(* IEC 61131-3 sources: elnaProjects/ElpcLogic/PomarKc7Changed/build_USO_ecl (part 7) *)

  fb_timer240(StrPh:=timer240);
  fb_PnmMore50(StrPh:=pmsMore50);
  fb_PnsOn(StrPh:=pnsOn, IM := Im.pns);
  fb_PmsMore300(StrPh:=pmsMore300);
  fb_Protection_Pms(StrPh:=Protection_Pms);
  fb_Error_Alg(StrPh:=Error_Alg);

  StrAlg.CanRun := StrAlg.inCanRun;
  StrAlg.OpcCommandsDisabled := StrAlg.inOpcCommandsDisabled;

  IF StrAlg.isRuning THEN

      StrAlg.hasError := pnsOn.error;

      (* не взведены защиты - запуск таймера *)
      IF NOT Protection_Pms.top THEN
  	runPhase(timer240);
      END_IF;

      (* не начался запуск пнс - запуск пнс *)
      IF NOT pnsOn.start THEN
  	runPhase(pnsOn);
      END_IF;

      (* запуск пнс завершен - запус защит *)
      IF pnsOn.top THEN
           runPhase(pmsMore50);
           runPhase(pmsMore300);
      END_IF;

      (* не завершился запуск защиты 50 - проверка давления 50 *)
      IF pmsMore50.start AND (NOT pmsMore50.top) THEN
  	IF ai.Pmaslo_sm_nizkoe.interval = _statusAi.NORMAL AND ai.Pmaslo_sm_nizkoe.value > 50.0  THEN
  	   pmsMore50.top := TRUE;
            END_IF;
      END_IF;

      (* не завершился запуск защиты 300 - проверка давления 300 *)
      IF  pmsMore300.start AND (NOT pmsMore300.top) THEN
  	IF ai.Pmaslo_sm_vysokoe.interval = _statusAi.NORMAL AND ai.Pmaslo_sm_vysokoe.value > 300.0  THEN
  	    pmsMore300.top := TRUE;
  	END_IF;
      END_IF;

      (* давление было проверено - запуск защит *)
      IF pmsMore50.top AND pmsMore300.top THEN
          runPhase(Protection_Pms);
      END_IF;

      (* запуск защит не завршен - запуск защит *)
      IF Protection_Pms.start AND (NOT Protection_Pms.top) THEN
  	runAiProtection(protections.Pmaslo_sm_nizkoe);
            runAiProtection(protections.Pmaslo_sm_vysokoe);
            Protection_Pms.top := TRUE;
      END_IF;

      (* таймер завершился до запуска защит - ошибка *)
      IF timer240.top THEN
          Error_Alg.ERROR := TRUE; (*не понятное куда его сунуть и нужен ли он*)
      ELSE
          Error_Alg.ERROR := FALSE;
      END_IF;

      (* защиты выствалены до завршения таймера - сброс таймера *)
      IF Protection_Pms.top THEN
  	resetPhase(timer240);
      END_IF;

      StrAlg.isEnded:= pnsOn.Top AND Protection_Pms.Top (*Как будто нужно таймер *);
  END_IF;

  StrAlg.CanRun := StrAlg.inCanRun;
  StrAlg.OpcCommandsDisabled := StrAlg.inOpcCommandsDisabled;

  (* ---- Если управление с ВУ заблокировано, то  передаем команду из алгоритма ---- *)
  IF StrAlg.inOpcCommandsDisabled THEN
  	StrAlg.inCommand := StrAlg.inCommand_Alg;
  ELSE (* иначе передаем команду с АРМа*)
  	StrAlg.inCommand := StrAlg.inCommand_ARM;
  END_IF;

  _sunpackerCommand(command := StrAlg.inCommand);
  	source := _sunpackerCommand.source;
  	cmd := _sunpackerCommand.cmd;

  IF cmd <> 0 AND lastCmd <> cmd AND (((NOT StrAlg.opcCommandsDisabled) AND source > 0) OR source = 0) then
  	CASE BYTE_TO_INT(cmd) OF
  		(*cmdRun*) 1: 	IF (StrAlg.CanRun) THEN
  					StrAlg.isRuning := TRUE;
  					StrAlg.isEnded := FALSE;
  					StrAlg.hasError := FALSE;
  					(*****************       OnRun       *****************)
                                                    algManager.nMode:=ModeGpa.MODE_PUSK_FIRST_FAZA1;

                                                    runPhase(pnsOn);
                                                    resetAiProtection(protections.Pmaslo_sm_nizkoe);
                                                    resetAiProtection(protections.Pmaslo_sm_vysokoe);

  					cmd_for_Status := cmd;
  					source_for_Status := source;
  					command_error_for_Status := 0;
  				ELSE
  					StrAlg.isRuning := FALSE;
  					StrAlg.isEnded := FALSE;
  					StrAlg.hasError := FALSE;

  					cmd_for_Status := 0;
  					source_for_Status := source;
  					command_error_for_Status := cmd;
  				END_IF;
  		(*cmdReset*) 2: 	StrAlg.isRuning := FALSE;
  				StrAlg.isEnded := FALSE;
  				StrAlg.hasError 	:= FALSE;

                                           (*****************       OnReset       *****************)
                                          waitReset(IN:=FALSE);
                                          StrAlg.inCanRun:=FALSE;

                                          resetPhase(timer240);
                                          resetPhase(pmsMore50);
                                          resetPhase(pnsOn);
                                          resetPhase(pmsMore300);
                                          resetPhase(Protection_Pms);
                                          resetPhase(Error_Alg);

                                          StrAlg.inOpcCommandsDisabled:=FALSE;

  				cmd_for_Status := cmd;
  				source_for_Status := source;
  				command_error_for_Status := 0;
  	END_CASE;
  	resetCmdTimer(IN := false);
  	resetCmdTimerPriznak := TRUE;
  END_IF;
  lastCmd := cmd;

  resetCmdTimer(IN := resetCmdTimerPriznak, PT := T#5S);
  IF resetCmdTimer.Q THEN
  	resetCmdTimerPriznak := FALSE;
  	source_for_Status := 0;
  	cmd_for_Status := 0;
  	command_error_for_Status := 0;
  END_IF;

  StrAlg.Start:= timer240.startStatus
              OR pmsMore50.startStatus
              OR pnsOn.startStatus
              OR Error_Alg.startStatus
              OR pmsMore300.startStatus
              OR Protection_Pms.startStatus;

  StrAlg.Error := timer240.errorStatus
              OR pmsMore50.errorStatus
              OR pnsOn.errorStatus
              OR Error_Alg.errorStatus
              OR pmsMore300.errorStatus
              OR Protection_Pms.errorStatus;

  StrAlg.Top := timer240.topStatus
              OR pmsMore50.topStatus
              OR pnsOn.topStatus
              OR Error_Alg.topStatus
              OR pmsMore300.topStatus
              OR Protection_Pms.topStatus;

  (*TODO: TYPE PROGRAM CODE HERE*)
  StrAlg.status :=  SHL(BYTE_TO_DWORD(source_for_Status), 29)
  			OR SHL(BYTE_TO_DWORD(cmd_for_Status), 26)
  			OR SHL(BYTE_TO_DWORD(command_error_for_Status), 23)
  			OR SHL(BOOL_TO_DWORD(StrAlg.OpcCommandsDisabled ), 21)
  			OR SHL(BOOL_TO_DWORD(StrAlg.hasError),4)
  			OR SHL(BOOL_TO_DWORD(StrAlg.CanRun),2)
  			OR SHL(BOOL_TO_DWORD(StrAlg.isEnded),1)
  			OR BOOL_TO_DWORD(StrAlg.isRuning);
END_FUNCTION_BLOCK

FUNCTION_BLOCK Prov_PMS
  VAR_IN_OUT
    StrAlg : struct_Alg;
  END_VAR
  VAR
    pnsOff : struct_PhaseAlgoritm;
    timer120 : struct_PhaseAlgoritm;
    Pms_less_25 : struct_PhaseAlgoritm;
    Pms_less_250 : struct_PhaseAlgoritm;
    Error_Alg : struct_PhaseAlgoritm;
    fb_Pms_less_25 : fb_ph_algoritm;
    fb_Pms_less_250 : fb_ph_algoritm;
    fb_pnsOff : fb_ph_Switch;
    fb_timer120 : fb_ph_Timer;
    fb_Error_Alg : fb_ph_algoritm;
    onInit : BOOL;
  END_VAR
  VAR_EXTERNAL
    Im : ImConfig;
    ai : AiConfig;
  END_VAR
  VAR
    _sunpackerCommand : fb_sunpackerCommand;
    source : BYTE;
    cmd : BYTE;
    _statusDualInput : TYPE_statusDualInput;
    lastCmd : BYTE;
    _Answers : TYPE_Answers;
  END_VAR
  VAR_EXTERNAL
    ModeGpa : TYPE_ModeGpa;
    algManager : struct_AlgoritmsManager;
  END_VAR
  VAR
    cmd_for_Status : BYTE;
    source_for_Status : BYTE;
    command_error_for_Status : BYTE;
    resetCmdTimer : TON;
    waitReset : TON;
    resetCmdTimerPriznak : BOOL;
    _statusAi : TYPE_StatusAi;
  END_VAR

  IF NOT onInit THEN
      fb_pnsOff(phaseNumber:=1, act:=_off);
      fb_timer120(phaseNumber:=2, delay:=T#120S);
      fb_Pms_less_25(phaseNumber:=3);
      fb_Pms_less_250(phaseNumber:=4);
      fb_Error_Alg(phaseNumber:=5);
      onInit:=TRUE;
  END_IF;

  fb_pnsOff(StrPh:=pnsOff, Im:=Im.pns);
  fb_timer120(StrPh:=timer120);
  fb_Pms_less_25(StrPh:=Pms_less_25);
  fb_Pms_less_250(StrPh:=Pms_less_250);
  fb_Error_Alg(StrPh:=Error_Alg);

  StrAlg.CanRun := StrAlg.inCanRun;
  StrAlg.OpcCommandsDisabled := StrAlg.inOpcCommandsDisabled;

  IF StrAlg.isRuning THEN
     (*IF NOT pnsOff.start THEN
  	    PNS_OFF_Ask.ask ();
      END_IF;
      IF	(PNS_OFF_Ask.answer=Answers.ANS_YES) THEN
  	    runPhase(pnsOff);
          PNS_OFF_Ask.reset ();
  	    IF NOT (Pms_less_250.top AND Pms_less_25.top) THEN
  	    	runPhase(timer120);
  	    END_IF;
      END_IF;*)

      (*запуск проверок давления*)
      IF	pnsOff.top  THEN
          runPhase(Pms_less_25);
  	    runPhase(Pms_less_250);
      END_IF;

      (*проверка давления масла низкое*)
      IF	Pms_less_25.start AND NOT Pms_less_25.top THEN
  	    IF 	ai.Pmaslo_sm_nizkoe.interval>=_statusAi.NORMAL AND ai.Pmaslo_sm_nizkoe.value < 25.0 THEN
  	  	    Pms_less_25.top:=TRUE;
  	    END_IF;
      END_IF;

      IF	Pms_less_250.start AND NOT Pms_less_250.top THEN
  	    IF	ai.Pmaslo_sm_vysokoe.interval>=_statusAi.NORMAL AND ai.Pmaslo_sm_vysokoe.value < 250.0 THEN
  	  	    Pms_less_250.top:=TRUE;
  	    END_IF;
      END_IF;

      (*ошибка заврешия алгоритма по таймеру*)
      IF	timer120.top THEN
  	    Error_Alg.ERROR := TRUE;
      ELSE
  	    Error_Alg.ERROR := FALSE;
      END_IF;

      (*если проверка прошла - сброс таймера *)
      IF	Pms_less_250.top AND Pms_less_25.top  THEN
          resetPhase(timer120);
      END_IF;
  END_IF;

  _sunpackerCommand(command := StrAlg.inCommand);
  	source := _sunpackerCommand.source;
  	cmd := _sunpackerCommand.cmd;

  IF cmd <> 0 AND lastCmd <> cmd AND (((NOT StrAlg.opcCommandsDisabled) AND source > 0) OR source = 0) then
  	CASE BYTE_TO_INT(cmd) OF
  		(*cm dRun*) 1: 	IF (StrAlg.CanRun) THEN
  					StrAlg.isRuning := TRUE;
  					StrAlg.isEnded := FALSE;
  					StrAlg.hasError := FALSE;
  					(*****************       OnRun       *****************)
                                                    algManager.nMode:=ModeGpa.MODE_PUSK_FIRST_FAZA2;

                                                    (*runPhase(timer120);
                                                    runPhase(timer5);
                                                    runPhase(Shup);
                                                    resetAiProtection(protections.dPmaslo_gaz);
                                                    resetDiProtection(protections.dPmaslo_gaz_less100);*)

  					cmd_for_Status := cmd;
  					source_for_Status := source;
  					command_error_for_Status := 0;
  				ELSE
  					StrAlg.isRuning := FALSE;
  					StrAlg.isEnded := FALSE;
  					StrAlg.hasError := FALSE;

  					cmd_for_Status := 0;
  					source_for_Status := source;
  					command_error_for_Status := cmd;
  				END_IF;
  		(*cmdReset*) 2: 	StrAlg.isRuning := FALSE;
  				StrAlg.isEnded := FALSE;
  				StrAlg.hasError 	:= FALSE;

                                           (*****************       OnReset       *****************)
                                          waitReset(IN:=FALSE);
                                          StrAlg.inCanRun:=FALSE;

                                          (*resetPhase(timer5);
                                          resetPhase(Shup);
                                          resetPhase(timer120);
                                          resetPhase(Net_Chast);
                                          resetPhase(mvOn);
                                          resetPhase(pGNSmore04);
                                          resetPhase(gotov_K_zagruzke);
                                          resetPhase(dPmg_Top);
                                          resetPhase(AutoPNS_Start);*)

                                          StrAlg.inOpcCommandsDisabled:=FALSE;

  				cmd_for_Status := cmd;
  				source_for_Status := source;
  				command_error_for_Status := 0;
  	END_CASE;
  	resetCmdTimer(IN := false);
  	resetCmdTimerPriznak := TRUE;
  END_IF;
  lastCmd := cmd;

  resetCmdTimer(IN := resetCmdTimerPriznak, PT := T#5S);
  IF resetCmdTimer.Q THEN
  	resetCmdTimerPriznak := FALSE;
  	source_for_Status := 0;
  	cmd_for_Status := 0;
  	command_error_for_Status := 0;
  END_IF;

  StrAlg.Start:= pnsOff.startStatus
              OR timer120.startStatus
              OR Pms_less_25.startStatus
              OR Pms_less_250.startStatus;

  StrAlg.Top :=  pnsOff.topStatus
              OR timer120.topStatus
              OR Pms_less_25.topStatus
              OR Pms_less_250.topStatus;

  StrAlg.Error :=  pnsOff.errorStatus
              OR timer120.errorStatus
              OR Pms_less_25.errorStatus
              OR Pms_less_250.errorStatus;

  (*TODO: TYPE PROGRAM CODE HERE*)
  StrAlg.status :=  SHL(BYTE_TO_DWORD(source_for_Status), 29)
  			OR SHL(BYTE_TO_DWORD(cmd_for_Status), 26)
  			OR SHL(BYTE_TO_DWORD(command_error_for_Status), 23)
  			OR SHL(BOOL_TO_DWORD(StrAlg.OpcCommandsDisabled ), 21)
  			OR SHL(BOOL_TO_DWORD(StrAlg.hasError),4)
  			OR SHL(BOOL_TO_DWORD(StrAlg.CanRun),2)
  			OR SHL(BOOL_TO_DWORD(StrAlg.isEnded),1)
  			OR BOOL_TO_DWORD(StrAlg.isRuning);
END_FUNCTION_BLOCK

FUNCTION_BLOCK Prov_opressovka
  VAR_IN_OUT
    StrAlg : struct_Alg;
  END_VAR
  VAR
    OPC_Control : struct_PhaseAlgoritm;
    Pms_more_50 : struct_PhaseAlgoritm;
    Pms_more_300 : struct_PhaseAlgoritm;
    dPmg_more_100 : struct_PhaseAlgoritm;
    P_zad : struct_PhaseAlgoritm;
    kran5Open : struct_PhaseAlgoritm;
    kran4Open : struct_PhaseAlgoritm;
    kran5Close : struct_PhaseAlgoritm;
    kran4Close : struct_PhaseAlgoritm;
    timer10 : struct_PhaseAlgoritm;
    P_vh_vyh_more_zad : struct_PhaseAlgoritm;
    Zapoln_Norm : struct_PhaseAlgoritm;
    First_Step : struct_PhaseAlgoritm;
    MaxZapolnenie_izm : REAL;
    Opressovka_Start : struct_Question;
    PNS_NU_ON_Ask : struct_Question;
    Zapolnit_kontur : struct_Question;
    fb_OPC_Control : fb_ph_algoritm;
    fb_Pms_more_50 : fb_ph_algoritm;
    fb_Pms_more_300 : fb_ph_algoritm;
    fb_dPmg_more_100 : fb_ph_algoritm;
    fb_P_zad : fb_ph_algoritm;
    fb_kran5Open : fb_ph_Kran;
    fb_kran4Open : fb_ph_Kran;
    fb_kran5Close : fb_ph_Kran;
    fb_kran4Close : fb_ph_Kran;
    fb_timer10 : fb_ph_Timer;
    fb_P_vh_vyh_more_zad : fb_ph_algoritm;
    fb_Zapoln_Norm : fb_ph_algoritm;
    fb_First_Step : fb_ph_algoritm;
    fb_Opressovka_Start : fb_Question;
    fb_PNS_NU_ON_Ask : fb_Question;
    fb_Zapolnit_kontur : fb_Question;
    onInit : BOOL;
  END_VAR
  VAR_EXTERNAL
    Im : ImConfig;
    ai : AiConfig;
  END_VAR
  VAR
    _sunpackerCommand : fb_sunpackerCommand;
    source : BYTE;
    cmd : BYTE;
    _statusDualInput : TYPE_statusDualInput;
    lastCmd : BYTE;
    _Answers : TYPE_Answers;
  END_VAR
  VAR_EXTERNAL
    ModeGpa : TYPE_ModeGpa;
    algManager : struct_AlgoritmsManager;
  END_VAR
  VAR
    cmd_for_Status : BYTE;
    source_for_Status : BYTE;
    command_error_for_Status : BYTE;
    resetCmdTimer : TON;
    waitReset : TON;
    resetCmdTimerPriznak : BOOL;
    _statusAi : TYPE_StatusAi;
    protections : ProtectionsConfig;
  END_VAR

  IF NOT onInit THEN
      fb_OPC_Control(phaseNumber:=1);
      fb_Pms_more_50(phaseNumber:=2);
      fb_Pms_more_300(phaseNumber:=3);
      fb_dPmg_more_100(phaseNumber:=4);
      fb_P_zad(phaseNumber:=5);
      fb_kran5Open(phaseNumber:=6, act:=_on);
      fb_kran4Open(phaseNumber:=7, act:=_on);
      fb_kran5Close(phaseNumber:=8, act:=_off);
      fb_kran4Close(phaseNumber:=9, act:=_off);
      fb_timer10(phaseNumber:=10, delay:=T#10S);
      fb_P_vh_vyh_more_zad(phaseNumber:=11);
      fb_Zapoln_Norm(phaseNumber:=12);
      fb_First_Step(phaseNumber:=13);
      Opressovka_Start.AnswerVariants:=_Answers.ANS_YES + _Answers.ANS_NO;
      PNS_NU_ON_Ask.AnswerVariants:=_Answers.ANS_YES;
      Zapolnit_kontur.AnswerVariants:=_Answers.ANS_YES;
      onInit:=TRUE;
  END_IF;

  fb_OPC_Control(StrPh:=OPC_Control);
  fb_Pms_more_50(StrPh:=Pms_more_50);
  fb_Pms_more_300(StrPh:=Pms_more_300);
  fb_dPmg_more_100(StrPh:=dPmg_more_100);
  fb_P_zad(StrPh:=P_zad);
  fb_kran5Open(StrPh:=kran5Open, Im:=Im.Kran5);
  fb_kran4Open(StrPh:=kran4Open, Im:=Im.Kran4);
  fb_kran5Close(StrPh:=kran5Close, Im:=Im.Kran5);
  fb_kran4Close(StrPh:=kran4Close, Im:=Im.Kran4);
  fb_timer10(StrPh:=timer10);
  fb_P_vh_vyh_more_zad(StrPh:=P_vh_vyh_more_zad);
  fb_Zapoln_Norm(StrPh:=Zapoln_Norm);
  fb_First_Step(StrPh:=First_Step);
  fb_Opressovka_Start(StrQ:=Opressovka_Start);
  fb_PNS_NU_ON_Ask(StrQ:=PNS_NU_ON_Ask);
  fb_Zapolnit_kontur(StrQ:=Zapolnit_kontur);

  StrAlg.CanRun := StrAlg.inCanRun;
  StrAlg.OpcCommandsDisabled := StrAlg.inOpcCommandsDisabled;

  IF StrAlg.isRuning THEN
     (*IF	algManager.mode <> ModeGpa.MODE_O THEN
  	    askQuestion(Opressovka_Start);
      END_IF;*)

      IF	Opressovka_Start.answer=_Answers.ANS_YES THEN
  	    askQuestion(Opressovka_Start);
  	    Im.kran6.inOpcCommandsDisabled := FALSE;
  	    (*algManager.setMode(nMode:=ModeGpa.MODE_O);*)
  	    runPhase(OPC_Control);
  	    resetAiProtection(protections.Pgaza_na_vyhode_nagnetatelia_GPA_STOP);
  	    resetAiProtection(protections.Pgaza_na_vhode_nagnetatelia_GPA_STOP);
          ELSIF Opressovka_Start.answer=_Answers.ANS_no THEN
                resetQuestion(Opressovka_Start);
      END_IF;

      IF	OPC_Control.start AND NOT OPC_Control.top THEN
  	    askQuestion(PNS_NU_ON_Ask);
      END_IF;
      IF	(PNS_NU_ON_Ask.answer=_Answers.ANS_YES) AND NOT OPC_Control.top THEN
  	    OPC_Control.top:=TRUE;
  	    resetQuestion(PNS_NU_ON_Ask);
      END_IF;

      IF	OPC_Control.top AND NOT Pms_more_50.start  THEN
  	    Im.pns.inOpcCommandsDisabled := FALSE;
  	    Im.kran6.inOpcCommandsDisabled := FALSE;
  	    runPhase(Pms_more_50);
  	    runPhase(Pms_more_300);
      END_IF;
      IF	OPC_Control.top AND Im.pns.onStatus = _statusDualInput.STATUS_On AND NOT dPmg_more_100.start THEN
  	    Im.nu1.inOpcCommandsDisabled := FALSE;
  	    Im.nu2.inOpcCommandsDisabled := FALSE;
  	    runPhase(dPmg_more_100);
      END_IF;

      IF	Im.nu1.onStatus = _statusDualInput.STATUS_On OR Im.nu2.onStatus = _statusDualInput.STATUS_On AND dPmg_more_100.start AND NOT dPmg_more_100.top THEN
  	    IF ai.dPmaslo_gaz.interval	>=	_statusAi.NORMAL AND
  		    ai.dPmaslo_gaz.value > 150.0 AND Im.SingleSignals.dP_maslo_gaz_Less100.reliability = TRUE AND NOT Im.SingleSignals.dP_maslo_gaz_Less100.Q THEN
  		    dPmg_more_100.top:=TRUE;
  		    runAiProtection(protections.dPmaslo_gaz);
  		    runDiProtection(protections.dPmaslo_gaz_less100);
  	    END_IF;
      END_IF;

      IF	Im.pns.onStatus = _statusDualInput.STATUS_On AND Pms_more_50.start AND NOT Pms_more_50.top THEN
  	        IF	ai.Pmaslo_sm_nizkoe.interval	>=	_statusAi.NORMAL AND
  		        ai.Pmaslo_sm_nizkoe.value > 50.0 THEN
  		        Pms_more_50.top:=TRUE;
                  runAiProtection(protections.Pmaslo_sm_nizkoe);
  	    END_IF;
      END_IF;

      IF	Im.pns.onStatus = _statusDualInput.STATUS_On AND Pms_more_300.start AND NOT Pms_more_300.top THEN
  	    IF	ai.Pmaslo_sm_vysokoe.interval	>=	_statusAi.NORMAL AND
  		    ai.Pmaslo_sm_vysokoe.value > 300.0 THEN
  		    Pms_more_300.top:=TRUE;
  		    runAiProtection(protections.Pmaslo_sm_vysokoe);
  	    END_IF;
      END_IF;

      (*IF	dPmg_more_100.top AND Pms_more_50.top AND Pms_more_300.top THEN
  	    CASE	Auto.value OF
  	    0:	Im.kran3.inOpcCommandsDisabled := FALSE;
  		Im.kran4.inOpcCommandsDisabled := FALSE;
  		Im.kran5.inOpcCommandsDisabled := FALSE;
  		Im.kran3b.inOpcCommandsDisabled := FALSE;
  		resetPhase(Zapolnit_kontur);
  		IF	Im.PerepadDavlenieKran1_Less100.Q THEN
  			Im.kran1.inOpcCommandsDisabled := FALSE;
  			Im.kran2.inOpcCommandsDisabled := FALSE;
  		ELSE
  			Im.kran1.inOpcCommandsDisabled := TRUE;
  			Im.kran2.inOpcCommandsDisabled := TRUE;
  		END_IF
  		resetPhase(P_vh_vyh_more_zad);
  		resetPhase(kran5Open);
  		resetPhase(kran4Open);
  		resetPhase(timer10);
  		resetPhase(kran5Close);
  		resetPhase(P_zad);
  		resetPhase(First_Step);
  		resetPhase(kran4Close);
  		(*MaxZapolnenie_izm:=0;
  		MaxZapolnenie.setValue (0);
  	1:
  		Zapoln_Norm.top:= MaxZapolnenie.value - MaxZapolnenie_izm > 0.4 AND MaxZapolnenie.value >= 0.4 AND MaxZapolnenie.value <= 10 AND
  			ai.DGazaNaVhodeNagnetatelja.interval >= _statusAi.NORMAL AND MaxZapolnenie.value - ai.DGazaNaVhodeNagnetatelja.value > 0.4 AND
  			ai.DGazaNaVyhodeNagnetatelja.interval >= _statusAi.NORMAL AND MaxZapolnenie.value - ai.DGazaNaVyhodeNagnetatelja.value > 0.4 *)
  		IF	kran4Close.top AND Zapoln_Norm.top AND NOT P_zad.start THEN
  			resetPhase(P_vh_vyh_more_zad);
  			resetPhase(kran5Open);
  			resetPhase(kran4Open);
  			resetPhase(timer10);
  			resetPhase(kran5Close);
  			resetPhase(kran4Close);
  		END_IF;
  		IF	NOT kran4Close.top OR kran4Close.top AND Zapoln_Norm.top AND NOT P_zad.start THEN
  		 	runPhase(P_zad);
  		END_IF;
  		IF NOT P_zad.top AND P_zad.start AND Zapoln_Norm.top THEN
  			askQuestion(Zapolnit_kontur);
  			Im.kran3.inOpcCommandsDisabled := TRUE;
  			Im.kran4.inOpcCommandsDisabled := TRUE;
  			Im.kran5.inOpcCommandsDisabled := TRUE;
  			Im.kran3b.inOpcCommandsDisabled := TRUE;
  			Im.kran1.inOpcCommandsDisabled := TRUE;
  			Im.kran2.inOpcCommandsDisabled := TRUE;

  		ELSIF NOT Zapoln_Norm.top AND NOT P_zad.top THEN
  				resetQuestion(Zapolnit_kontur);
  		END_IF;

          IF	(Zapolnit_kontur.answer=_Answers.ANS_YES) AND P_zad.start THEN
  			(*MaxZapolnenie_izm:= MaxZapolnenie.value;*)
  			IF 	NOT First_Step.top THEN
  				runPhase(kran5Open);
  			ELSE
  				runPhase(kran4Open);
  			END_IF;
  			resetQuestion(Zapolnit_kontur);
  			P_zad.top:=TRUE;
  		END_IF;
                      (*

  		IF	P_zad.top AND NOT kran4Close.top THEN
  			MaxZapolnenie.newvalue:=MaxZapolnenie_izm;
  		ELSE
  			MaxZapolnenie.newvalue:= MaxZapolnenie.newvalue;
  		END_IF;*)

  		IF	kran5Open.top AND NOT First_Step.top THEN
  			runPhase(kran4Open);
  		END_IF;

          IF 	kran4Open.top AND NOT timer10.top AND NOT First_Step.top THEN
  			runPhase(timer10);
  		END_IF;

  		IF	timer10.top AND NOT First_Step.top THEN
  			runPhase(kran5Close);
  		END_IF;

  		IF	kran5Close.top OR First_Step.top AND kran4Open.top THEN
  			runPhase(P_vh_vyh_more_zad);
          END_IF;

  		IF	ai.Pgaza_na_vhode_nagnetatelia.interval >= _statusAi.NORMAL (*AND ai.Pgaza_na_vhode_nagnetatelia.value >= MaxZapolnenie.value*) AND
  			ai.Pgaza_na_vyhode_nagnetatelia.interval >= _statusAi.NORMAL (*AND ai.Pgaza_na_vyhode_nagnetatelia.value >= MaxZapolnenie.value*) AND  P_vh_vyh_more_zad.start AND NOT P_vh_vyh_more_zad.top THEN
  			runPhase(kran4Close);
  			P_vh_vyh_more_zad.top:=TRUE;
  		END_IF;

  		IF	kran4Close.top THEN
  			First_Step.top:=TRUE;
  			Im.kran3.inOpcCommandsDisabled := FALSE;
  			Im.kran4.inOpcCommandsDisabled := FALSE;
  			Im.kran5.inOpcCommandsDisabled := FALSE;
  			Im.kran3b.inOpcCommandsDisabled := FALSE;

              IF	Zapoln_Norm.top THEN
  				resetPhase(P_zad);
  			END_IF;

              IF	Im.SingleSignals.dp_kran1_Less100.Q THEN
  				Im.kran1.inOpcCommandsDisabled := FALSE;
  				Im.kran2.inOpcCommandsDisabled := FALSE;
  			ELSE
  				Im.kran1.inOpcCommandsDisabled := TRUE;
  				Im.kran2.inOpcCommandsDisabled := TRUE;
  			END_IF;
  		ELSE
  			Im.kran1.inOpcCommandsDisabled := TRUE;
  			Im.kran2.inOpcCommandsDisabled := TRUE;
  	    END_IF;
          END_IF;
          (*END_CASE;
  END_IF;*)

  _sunpackerCommand(command := StrAlg.inCommand);
  	source := _sunpackerCommand.source;
  	cmd := _sunpackerCommand.cmd;

  IF cmd <> 0 AND lastCmd <> cmd AND (((NOT StrAlg.opcCommandsDisabled) AND source > 0) OR source = 0) then
  	CASE BYTE_TO_INT(cmd) OF
  		(*cm dRun*) 1: 	IF (StrAlg.CanRun) THEN
  					StrAlg.isRuning := TRUE;
  					StrAlg.isEnded := FALSE;
  					StrAlg.hasError := FALSE;
  					(*****************       OnRun       *****************)
                                                    algManager.nMode:=ModeGpa.MODE_PUSK_FIRST_FAZA2;

                                                    (*runPhase(timer120);
                                                    runPhase(timer5);
                                                    runPhase(Shup);
                                                    resetAiProtection(protections.dPmaslo_gaz);
                                                    resetDiProtection(protections.dPmaslo_gaz_less100);*)

  					cmd_for_Status := cmd;
  					source_for_Status := source;
  					command_error_for_Status := 0;
  				ELSE
  					StrAlg.isRuning := FALSE;
  					StrAlg.isEnded := FALSE;
  					StrAlg.hasError := FALSE;

  					cmd_for_Status := 0;
  					source_for_Status := source;
  					command_error_for_Status := cmd;
  				END_IF;
  		(*cmdReset*) 2: 	StrAlg.isRuning := FALSE;
  				StrAlg.isEnded := FALSE;
  				StrAlg.hasError 	:= FALSE;

                                           (*****************       OnReset       *****************)
                                          waitReset(IN:=FALSE);
                                          StrAlg.inCanRun:=FALSE;

                                          (*resetPhase(timer5);
                                          resetPhase(Shup);
                                          resetPhase(timer120);
                                          resetPhase(Net_Chast);
                                          resetPhase(mvOn);
                                          resetPhase(pGNSmore04);
                                          resetPhase(gotov_K_zagruzke);
                                          resetPhase(dPmg_Top);
                                          resetPhase(AutoPNS_Start);*)

                                          StrAlg.inOpcCommandsDisabled:=FALSE;

  				cmd_for_Status := cmd;
  				source_for_Status := source;
  				command_error_for_Status := 0;
  	END_CASE;
  	resetCmdTimer(IN := false);
  	resetCmdTimerPriznak := TRUE;
  END_IF;
  lastCmd := cmd;

  resetCmdTimer(IN := resetCmdTimerPriznak, PT := T#5S);
  IF resetCmdTimer.Q THEN
  	resetCmdTimerPriznak := FALSE;
  	source_for_Status := 0;
  	cmd_for_Status := 0;
  	command_error_for_Status := 0;
  END_IF;

  StrAlg.Start:= OPC_Control.startStatus
              OR Pms_more_50.startStatus
              OR Pms_more_300.startStatus
              OR dPmg_more_100.startStatus
              OR P_zad.startStatus
              OR kran5Open.startStatus
              OR kran4Open.startStatus
              OR kran5Close.startStatus
              OR kran4Close.startStatus
              OR timer10.startStatus
              OR P_vh_vyh_more_zad.startStatus
              OR Zapoln_Norm.startStatus
              OR First_Step.startStatus;

  StrAlg.Top :=  OPC_Control.topStatus
              OR Pms_more_50.topStatus
              OR Pms_more_300.topStatus
              OR dPmg_more_100.topStatus
              OR P_zad.topStatus
              OR kran5Open.topStatus
              OR kran4Open.topStatus
              OR kran5Close.topStatus
              OR kran4Close.topStatus
              OR timer10.topStatus
              OR P_vh_vyh_more_zad.topStatus
              OR Zapoln_Norm.topStatus
              OR First_Step.topStatus;

  StrAlg.Error :=  OPC_Control.errorStatus
              OR Pms_more_50.errorStatus
              OR Pms_more_300.errorStatus
              OR dPmg_more_100.errorStatus
              OR P_zad.errorStatus
              OR kran5Open.errorStatus
              OR kran4Open.errorStatus
              OR kran5Close.errorStatus
              OR kran4Close.errorStatus
              OR timer10.errorStatus
              OR P_vh_vyh_more_zad.errorStatus
              OR Zapoln_Norm.errorStatus
              OR First_Step.errorStatus;

  (*TODO: TYPE PROGRAM CODE HERE*)
  StrAlg.status :=  SHL(BYTE_TO_DWORD(source_for_Status), 29)
  			OR SHL(BYTE_TO_DWORD(cmd_for_Status), 26)
  			OR SHL(BYTE_TO_DWORD(command_error_for_Status), 23)
  			OR SHL(BOOL_TO_DWORD(StrAlg.OpcCommandsDisabled ), 21)
  			OR SHL(BOOL_TO_DWORD(StrAlg.hasError),4)
  			OR SHL(BOOL_TO_DWORD(StrAlg.CanRun),2)
  			OR SHL(BOOL_TO_DWORD(StrAlg.isEnded),1)
  			OR BOOL_TO_DWORD(StrAlg.isRuning);
END_FUNCTION_BLOCK

FUNCTION_BLOCK Pusk_second_faza_chastotny
  VAR_IN_OUT
    StrAlg : struct_Alg;
  END_VAR
  VAR
    timer120 : struct_PhaseAlgoritm;
    timer5 : struct_PhaseAlgoritm;
    Shup : struct_PhaseAlgoritm;
    Net_Chast : struct_PhaseAlgoritm;
    mvOn : struct_PhaseAlgoritm;
    pGNSmore04 : struct_PhaseAlgoritm;
    gotov_K_zagruzke : struct_PhaseAlgoritm;
    dPmg_Top : struct_PhaseAlgoritm;
    AutoPNS_Start : struct_PhaseAlgoritm;
    fb_timer120 : fb_ph_Timer;
    fb_timer5 : fb_ph_Timer;
    fb_Shup : fb_ph_OilPump;
    fb_Net_Chast : fb_ph_algoritm;
    fb_mvOn : fb_ph_SectionSwitch;
    fb_pGNSmore04 : fb_ph_algoritm;
    fb_gotov_K_zagruzke : fb_ph_algoritm;
    fb_dPmg_Top : fb_ph_algoritm;
    fb_AutoPNS_Start : fb_ph_algoritm;
    _sunpackerCommand : fb_sunpackerCommand;
    _statusDualInput : TYPE_statusDualInput;
    _Answers : TYPE_Answers;
    source : BYTE;
    cmd : BYTE;
    lastCmd : BYTE;
    source_for_Status : BYTE;
    cmd_for_Status : BYTE;
    command_error_for_Status : BYTE;
    resetCmdTimer : TON;
    resetCmdTimerPriznak : BOOL;
    onInit : BOOL;
    waitReset : TON;
  END_VAR
  VAR_EXTERNAL
    ModeGpa : TYPE_ModeGpa;
    algManager : struct_AlgoritmsManager;
    IM : ImConfig;
    protections : ProtectionsConfig;
    algoritms : AlgoritmsConfig;
    ai : AiConfig;
  END_VAR
  VAR
    statusAi : TYPE_StatusAi;
  END_VAR

  IF NOT onInit THEN
           fb_timer120(phaseNumber:=1, delay:=T#120S);
           fb_timer5(phaseNumber:=2, delay:=T#5S);
           fb_Shup(phaseNumber:=3);
           fb_Net_Chast(phaseNumber:=4);
           fb_mvOn(phaseNumber:=5,  act:=_on);
           fb_pGNSmore04(phaseNumber:=6);
           fb_gotov_K_zagruzke(phaseNumber:=7);
           fb_dPmg_Top(phaseNumber:=8);
           fb_AutoPNS_Start(phaseNumber:=9, act:=_run, waitCompletion:=FALSE);
  onInit:=TRUE;
  END_IF;

  fb_timer120(StrPh:=timer120);
  fb_timer5(StrPh:= timer5);
  fb_Shup(StrPh:= Shup);
  fb_Net_Chast(StrPh:=Net_Chast);
  fb_mvOn(StrPh:=mvOn, Im:=IM.mv);
  fb_pGNSmore04(StrPh:=pGNSmore04);
  fb_gotov_K_zagruzke(StrPh:=gotov_K_zagruzke);
  fb_dPmg_Top(StrPh:=dPmg_Top);
  fb_AutoPNS_Start(StrPh:=AutoPNS_Start, alg:=algoritms.autoPns);

  StrAlg.CanRun := StrAlg.inCanRun;
  StrAlg.OpcCommandsDisabled := StrAlg.inOpcCommandsDisabled;

  IF StrAlg.isRuning THEN
      (* мв не включен - запуск таймера *)
      IF NOT mvOn.top THEN
  	runphase(timer120);
      END_IF;
      (* частотный пуск не совершен - запуск таймера *)
      IF NOT Net_Chast.top THEN
  	runphase(timer5);
      END_IF;

      (* ШУП не запущен - запуск *)
      IF NOT Shup.start THEN
  	runphase(Shup);
      END_IF;

      (* ШУП не завершился - запуск ШУПб МВ *)
      IF NOT Shup.top AND Shup.start THEN
  	runIfNotRunningSO(IM.SingleOutputs.Pusk_SHUP);
  	Shup.top:=TRUE;
  	runphase(mvOn);
      END_IF;

      (* частотный пуск не запущен - запуск *)
      IF NOT Net_Chast.start THEN
  	runphase(Net_Chast);
      END_IF;

      (* частотный пуск не завершился - запуск *)
      IF Net_Chast.start AND (NOT Net_Chast.top) THEN
  	IF (NOT IM.SingleSignals.Chastotny_pusk.Q) AND (IM.SingleSignals.Chastotny_pusk.status = 1) THEN
  		Net_Chast.top:=TRUE;
  		resetPhase(timer5);
  	END_IF;
      END_IF;

      (* таймер не истек и мв не включен - вовзедение защиты *)
      IF (NOT timer120.top) AND (NOT mvOn.top) THEN
  	runDiProtection(protections.Fail_chastotnii_pusk);
      ELSE
  	resetDiProtection(protections.Fail_chastotnii_pusk);
      END_IF;

      (* мв не завершился - включение мв *)
      IF mvOn.start AND NOT mvOn.top THEN
  	IF IM.mv.onStatus = _statusDualInput.STATUS_ON THEN
                mvOn.top:=TRUE;
  	END_IF;
      END_IF;

      (* мв завершился - что-то делаем *)
      IF mvOn.top THEN
  	IF NOT pGNSmore04.start (*AND (algManager.mode = ModeGpa.MODE_PUSKPP_Ch OR algManager.mode = ModeGpa.MODE_PUSKAP_Ch)какой режим *) THEN
  		runphase(pGNSmore04);
  	END_IF;
           (* IF NOT autoAVOM_canrun_flag THEN
                algoritms.AutoAvom.CanRun:=TRUE;
  	    autoAVOM_canrun_flag:=TRUE; kto ti
  	END_IF;*)
  	resetPhase(timer120);
  	runphase(gotov_K_zagruzke);

            IF NOT dPmg_Top.start (* AND ((algManager.mode = modegpa.MODE_PUSKAP_Ch) OR (algManager.mode = modegpa.MODE_PUSKPP_Ch))*) THEN
                runphase(dPmg_Top);
  	END_IF;

            runAiProtection(protections.Pgaza_na_vyhode_nagnetatelia_GPA_STOP);
  	runDiProtection(protections.Off_avar_vikluchatel);
  	runDiProtection(protections.Reg_vozb_off);
      END_IF;

      IF dPmg_Top.start AND NOT dPmg_Top.top THEN
  	IF NOT IM.SingleSignals.dP_maslo_gaz_Less100.Q AND IM.SingleSignals.dP_maslo_gaz_Less100.status = 1 AND ai.dPmaslo_gaz.value > 150.0 THEN
  		dPmg_Top.top:=TRUE;
  		runAiProtection(protections.dPmaslo_gaz);
  		runDiProtection(protections.dPmaslo_gaz_less100);
  		resetAiProtection(protections.Pgaza_na_vhode_nagnetatelia_GPA_STOP);
  		resetAiProtection(protections.Pgaza_na_vyhode_nagnetatelia_GPA_STOP);
  		algoritms.autoNu.CanRun:=TRUE;
  		(*algoritms.autoNu.run(); кого чего, ничего не понимаю *)
  	END_IF;
      END_IF;

      IF pGNSmore04.start AND NOT pGNSmore04.top THEN
  	IF ai.Pmasla_posle_GNS.interval (*почему интервал, если есть статус *) >= statusAi.NORMAL AND ai.Pmasla_posle_GNS.value > 400.0 THEN
  	  	pGNSmore04.top:=TRUE;
  	END_IF;
      END_IF;

      IF (pGNSmore04.top AND gotov_K_zagruzke.top AND dPmg_Top.top )(*AND (algManager.mode = modegpa.MODE_PUSKAP_Ch OR (algManager.mode = modegpa.MODE_PUSKPP_Ch) *)OR
  	(gotov_K_zagruzke.top) (*AND (algManager.mode = modegpa.MODE_PUSKV_Ch OR algManager.mode = modegpa.MODE_I))*) AND NOT AutoPNS_Start.top  THEN
  	algoritms.AutoPns.CanRun :=TRUE;
  	(*algoritms.AutoPns;*)
  	AutoPNS_Start.top:=TRUE;
      END_IF;

      IF (NOT Net_Chast.top AND timer5.top) OR (timer120.top AND NOT mvOn.top) THEN
  	algoritms.ao.CanRun:=TRUE;
  	(*algoritms.ao.run ();*)
      END_IF;
  END_IF;

  StrAlg.CanRun := StrAlg.inCanRun;
  StrAlg.OpcCommandsDisabled := StrAlg.inOpcCommandsDisabled;

  (* ---- Если управление с ВУ заблокировано, то  передаем команду из алгоритма ---- *)
  IF StrAlg.inOpcCommandsDisabled THEN
  	StrAlg.inCommand := StrAlg.inCommand_Alg;
  ELSE (* иначе передаем команду с АРМа*)
  	StrAlg.inCommand := StrAlg.inCommand_ARM;
  END_IF;

  _sunpackerCommand(command := StrAlg.inCommand);
  	source := _sunpackerCommand.source;
  	cmd := _sunpackerCommand.cmd;

  IF cmd <> 0 AND lastCmd <> cmd AND (((NOT StrAlg.opcCommandsDisabled) AND source > 0) OR source = 0) then
  	CASE BYTE_TO_INT(cmd) OF
  		(*cmdRun*) 1: 	IF (StrAlg.CanRun) THEN
  					StrAlg.isRuning := TRUE;
  					StrAlg.isEnded := FALSE;
  					StrAlg.hasError := FALSE;
  					(*****************       OnRun       *****************)
                                                    algManager.nMode:=ModeGpa.MODE_PUSK_FIRST_FAZA2;

                                                    runPhase(timer120);
                                                    runPhase(timer5);
                                                    runPhase(Shup);
                                                    resetAiProtection(protections.dPmaslo_gaz);
                                                    resetDiProtection(protections.dPmaslo_gaz_less100);

  					cmd_for_Status := cmd;
  					source_for_Status := source;
  					command_error_for_Status := 0;
  				ELSE
  					StrAlg.isRuning := FALSE;
  					StrAlg.isEnded := FALSE;
  					StrAlg.hasError := FALSE;

  					cmd_for_Status := 0;
  					source_for_Status := source;
  					command_error_for_Status := cmd;
  				END_IF;
  		(*cmdReset*) 2: 	StrAlg.isRuning := FALSE;
  				StrAlg.isEnded := FALSE;
  				StrAlg.hasError 	:= FALSE;

                                           (*****************       OnReset       *****************)
                                          waitReset(IN:=FALSE);
                                          StrAlg.inCanRun:=FALSE;

                                          resetPhase(timer5);
                                          resetPhase(Shup);
                                          resetPhase(timer120);
                                          resetPhase(Net_Chast);
                                          resetPhase(mvOn);
                                          resetPhase(pGNSmore04);
                                          resetPhase(gotov_K_zagruzke);
                                          resetPhase(dPmg_Top);
                                          resetPhase(AutoPNS_Start);

                                          StrAlg.inOpcCommandsDisabled:=FALSE;

  				cmd_for_Status := cmd;
  				source_for_Status := source;
  				command_error_for_Status := 0;
  	END_CASE;
  	resetCmdTimer(IN := false);
  	resetCmdTimerPriznak := TRUE;
  END_IF;
  lastCmd := cmd;

  resetCmdTimer(IN := resetCmdTimerPriznak, PT := T#5S);
  IF resetCmdTimer.Q THEN
  	resetCmdTimerPriznak := FALSE;
  	source_for_Status := 0;
  	cmd_for_Status := 0;
  	command_error_for_Status := 0;
  END_IF;

  StrAlg.Start:= timer120.startStatus
              OR timer5.startStatus
              OR Shup.startStatus
              OR Net_Chast.startStatus
              OR mvOn.startStatus
              OR pGNSmore04.startStatus
              OR gotov_K_zagruzke.startStatus
              OR dPmg_Top.startStatus
              OR AutoPNS_Start.startStatus;

  StrAlg.Error := timer120.errorStatus
              OR timer5.errorStatus
              OR Shup.errorStatus
              OR Net_Chast.errorStatus
              OR mvOn.errorStatus
              OR pGNSmore04.errorStatus
              OR gotov_K_zagruzke.errorStatus
              OR dPmg_Top.errorStatus
              OR AutoPNS_Start.errorStatus;

  StrAlg.Top := timer120.topStatus
              OR timer5.topStatus
              OR Shup.topStatus
              OR Net_Chast.topStatus
              OR mvOn.topStatus
              OR gotov_K_zagruzke.topStatus
              OR dPmg_Top.topStatus
              OR AutoPNS_Start.topStatus
              OR pGNSmore04.topStatus;

  (*TODO: TYPE PROGRAM CODE HERE*)
  StrAlg.status :=  SHL(BYTE_TO_DWORD(source_for_Status), 29)
  			OR SHL(BYTE_TO_DWORD(cmd_for_Status), 26)
  			OR SHL(BYTE_TO_DWORD(command_error_for_Status), 23)
  			OR SHL(BOOL_TO_DWORD(StrAlg.OpcCommandsDisabled ), 21)
  			OR SHL(BOOL_TO_DWORD(StrAlg.hasError),4)
  			OR SHL(BOOL_TO_DWORD(StrAlg.CanRun),2)
  			OR SHL(BOOL_TO_DWORD(StrAlg.isEnded),1)
  			OR BOOL_TO_DWORD(StrAlg.isRuning);
END_FUNCTION_BLOCK

FUNCTION_BLOCK proc_algoritms
  VAR
    fb_RemontAlg : RemontAlg;
    fb_TestProtectionAlg : TestProtectionAlg;
    fb_TestImAlg : TestImAlg;
    fb_AutoTen : fb_AutoTenAlg;
    fb_AutoPns : fb_AutoPnsAlg;
    fb_AutoAvom : fb_AutoAvomAlg;
    fb_vibegPNS : fb_vibegPNSAlg;
    fb_AutoNU : fb_AutoNUAlg;
    fb_puskOilSystem : fb_puskOilSystemAlg;
    fb_AntiPompag : fb_AntiPompagAlg;
    fb_NOAlg : NOAlg;
    fb_AOAlg : AOAlg;
    fb_ppuALG : ppuAlg;
    fb_fillingAlg : fillingAlg;
    fb_engineRunAlg : engineRunAlg;
    fb_puskKalg : puskKalg;
    fb_puskValg : puskValg;
    fb_testdPmgAlg : testdPmgAlg;
    fb_testPmsAlg : testPmsAlg;
    fb_ApuskAlg : ApuskAlg;
    fb_SemiAutoPuskAlg : SemiAutoPuskAlg;
    fb_Pusk_first_faza1 : Pusk_first_faza1;
    fb_Pusk_first_faza2 : Pusk_first_faza2;
    fb_Pusk_third_faza : Pusk_third_faza;
    fb_Pusk_Prov_PMS : Prov_PMS;
    fb_Prov_opressovka : Prov_opressovka;
    fb_Pusk_second_faza_chastotny : Pusk_second_faza_chastotny;
    fb_Pusk_second_faza_reactor : Pusk_second_faza_reactor;
  END_VAR
  VAR_EXTERNAL
    algoritms : AlgoritmsConfig;
    AlgQuestions : AlgoritmsQuestions;
    ai : AiConfig;
    IM : ImConfig;
    AlgTimers : struct_AlgTimers;
  END_VAR

  fb_RemontAlg(StrAlg:=algoritms.Remont);

  fb_TestProtectionAlg(StrAlg:=algoritms.TestProtection);

  fb_TestImAlg(StrAlg:=algoritms.testIm);

  (*fb_AutoTen(StrAlg:= algoritms.AutoTen,
  T_masla:= ai.Toporno_podshipnika_EDT_1,
  Uroven_masla:= ai.Yroven_masla_MB,
  offTemperature:= Im.AutoTen_offTemperature,
  TEN:= Im.Ten,
  PNS:= Im.pns);*)

  (*fb_AutoPns(StrAlg:= algoritms.AutoPns,
  Poil:= ai.Pmasla_posle_GNS,
  Ust_Run:= Im.AutoPns_UstRun,
  Ust_Stop:= Im.AutoPns_UstStop,
  Nasos:= Im.pns,
  diPlow:= Im.SingleSignals.P_oil_low);*)

  (*fb_AutoAvom(StrAlg:= algoritms.AutoAvom,
  im1:= Im.v1_Avom,
  im2:= Im.v2_Avom,
  on1Temperature:= Im.AutoAvom_onTemp1,
  on2Temperature:= Im.AutoAvom_onTemp2,
  hystereses:= Im.AutoAvom_hysteresis,
  ai:= ai.Tnarujnogo_vozduha);*)

  fb_vibegPNS(StrAlg:=algoritms.vibegPNS,
  algContinue:=AlgQuestions.vibegPNS_algContinue
  );

  (*fb_AutoNU(StrAlg:=algoritms.autoNu,
  nu1:=Im.nu1,
  nu2:=Im.nu2,
  Ust_Swap:= Im.AutoNU_Ust_Swap,
  mainNU:= Im.AutoNU_mainNU,
  dPoil:=ai.Tmasla_MB,
  Lowdp_di:=Im.SingleSignals.dP_oilgaz_low
  );*)

  fb_puskOilSystem(StrAlg:=algoritms.puskOilSystem);

  (*fb_AntiPompag(StrAlg:=algoritms.AntiPompag,
  Rashod:= ai.Vibro_skorost_OP_shesterni_RED_T6,
  Zapas:= ai.Vibro_skorost_OP_shesterni_RED_T5,
  P_gasIn:=ai.dPgaza_na_maslo_filtre,
  T_gasIn:=ai.Tgaza_na_vhode_H,
  dP_konf:=ai.dPgaza_na_konfuzore,
  Kran6:= im.Kran6,
  UgolVNA:= im.AntiPompag_UgolVNA,
  K:=im.AntiPompag_K,
  A:=im.AntiPompag_A,
  y0:=im.AntiPompag_y0);*)

  fb_NOAlg(StrAlg:=algoritms.no);

  fb_AOAlg(StrAlg:=algoritms.ao);

  fb_ppuAlg(StrAlg:=algoritms.ppu);

  fb_fillingAlg(StrAlg:=algoritms.filling);

  fb_engineRunAlg(StrAlg:=algoritms.engineRun);

  fb_puskKalg(StrAlg:=algoritms.puskK,
  questionFilling:=AlgQuestions.puskK_questionFilling,
   questionUnload:=AlgQuestions.puskK_questionUnload
  );

  fb_puskValg(StrAlg:=algoritms.puskV,
   questionEngine:=AlgQuestions.puskV_questionEngine,
    questionMVoff:=AlgQuestions.puskV_questionMVoff
  );

  fb_testdPmgAlg(StrAlg:=algoritms.testdPmg,
   algContinue:=AlgQuestions.testdPmg_algContinue
  );

  fb_testPmsAlg(StrAlg:=algoritms.testPms,
   algContinue:=AlgQuestions.testPms_algContinue
  );

  fb_ApuskAlg(StrAlg:=algoritms.Apusk);

  fb_SemiAutoPuskAlg(StrAlg:=algoritms.SemiAutoPusk,
   cmdRun1ph:=AlgQuestions.SemiAutoPusk_cmdRun1ph,
   cmdRun2ph:=AlgQuestions.SemiAutoPusk_cmdRun2ph,
   cmdRun3ph:=AlgQuestions.SemiAutoPusk_cmdRun3ph
  );

  fb_Pusk_first_faza1(Stralg:=algoritms.Pusk_F_faza1);

  fb_Pusk_first_faza2(Stralg:=algoritms.Pusk_F_faza2);

  fb_Pusk_third_faza(Stralg:=algoritms.Pusk_TH_faza);

  fb_Pusk_Prov_PMS(Stralg:=algoritms.Prov_PMS_ALG);

  fb_Prov_opressovka(Stralg:=algoritms.Prov_opressovka_ALG);

  fb_Pusk_second_faza_chastotny(Stralg:=algoritms.Pusk_SEC_faza_chastotny);

  fb_Pusk_second_faza_reactor(Stralg:=algoritms.Pusk_SEC_faza_reactor);
END_FUNCTION_BLOCK

FUNCTION_BLOCK OPC_IM_GET
  VAR_EXTERNAL
    IM : ImConfig;
    IM_Kran1_status : UDINT;
    IM_Kran1_inCommand_ARM : UINT;
    IM_Kran2_status : UDINT;
    IM_Kran2_inCommand_ARM : UINT;
    IM_Kran3_status : UDINT;
    IM_Kran3_inCommand_ARM : UINT;
    IM_Kran3b_status : UDINT;
    IM_Kran3b_inCommand_ARM : UINT;
    IM_Kran4_status : UDINT;
    IM_Kran4_inCommand_ARM : UINT;
    IM_Kran5_status : UDINT;
    IM_Kran5_inCommand_ARM : UINT;
    IM_Kran6_status : UDINT;
    IM_Kran6_inCommand_ARM : UINT;
    IM_nu1_status : UDINT;
    IM_nu1_inCommand_ARM : UINT;
    IM_nu2_status : UDINT;
    IM_nu2_inCommand_ARM : UINT;
    IM_pns_status : UDINT;
    IM_pns_inCommand_ARM : UINT;
    IM_v1_Avom_status : UDINT;
    IM_v1_Avom_inCommand_ARM : UINT;
    IM_v2_Avom_status : UDINT;
    IM_v2_Avom_inCommand_ARM : UINT;
    IM_v3_Avom_status : UDINT;
    IM_v3_Avom_inCommand_ARM : UINT;
    IM_v4_Avom_status : UDINT;
    IM_v4_Avom_inCommand_ARM : UINT;
    IM_mv_status : UDINT;
    IM_mv_inCommand_ARM : UINT;
    IM_KaloriferAVOM_status : UDINT;
    IM_KaloriferAVOM_inCommand_ARM : UINT;
    IM_CMN_status : UDINT;
    IM_CMN_inCommand_ARM : UINT;
    IM_TEN_kollectora_status : UDINT;
    IM_TEN_kollectora_inCommand_ARM : UINT;
    IM_TEN_MB_status : UDINT;
    IM_TEN_MB_inCommand_ARM : UINT;
  END_VAR

  IM.Kran1.inCommand_ARM := UINT_TO_WORD(IM_Kran1_inCommand_ARM);

  IM.Kran2.inCommand_ARM := UINT_TO_WORD(IM_Kran2_inCommand_ARM);

  IM.Kran3.inCommand_ARM := UINT_TO_WORD(IM_Kran3_inCommand_ARM);

  IM.Kran3b.inCommand_ARM := UINT_TO_WORD(IM_Kran3b_inCommand_ARM);

  IM.Kran4.inCommand_ARM := UINT_TO_WORD(IM_Kran4_inCommand_ARM);

  IM.Kran5.inCommand_ARM := UINT_TO_WORD(IM_Kran5_inCommand_ARM);

  IM.Kran6.inCommand_ARM := UINT_TO_WORD(IM_Kran6_inCommand_ARM);

  IM.nu1.inCommand_ARM := UINT_TO_WORD(IM_nu1_inCommand_ARM);

  IM.nu2.inCommand_ARM := UINT_TO_WORD(IM_nu2_inCommand_ARM);

  IM.pns.inCommand_ARM := UINT_TO_WORD(IM_pns_inCommand_ARM);

  IM.v1_Avom.inCommand_ARM := UINT_TO_WORD(IM_v1_Avom_inCommand_ARM);

  IM.v2_Avom.inCommand_ARM := UINT_TO_WORD(IM_v2_Avom_inCommand_ARM);

  IM.v3_Avom.inCommand_ARM := UINT_TO_WORD(IM_v3_Avom_inCommand_ARM);

  IM.v4_Avom.inCommand_ARM := UINT_TO_WORD(IM_v4_Avom_inCommand_ARM);

  IM.mv.inCommand_ARM := UINT_TO_WORD(IM_mv_inCommand_ARM);

  IM.KaloriferAVOM.inCommand_ARM := UINT_TO_WORD(IM_KaloriferAVOM_inCommand_ARM);

  IM.CMN.inCommand_ARM := UINT_TO_WORD(IM_CMN_inCommand_ARM);

  IM.TEN_kollectora.inCommand_ARM := UINT_TO_WORD(IM_TEN_kollectora_inCommand_ARM);

  IM.TEN_MB.inCommand_ARM := UINT_TO_WORD(IM_TEN_MB_inCommand_ARM);
END_FUNCTION_BLOCK

FUNCTION_BLOCK OPC_algoritms_set
  VAR_EXTERNAL
    algoritms : AlgoritmsConfig;
    algManager_Mode : UINT;
    algoritms_AutoAvom_status : UDINT;
    algoritms_AutoPns_OffTimer : UINT;
    algoritms_AutoPns_OnTimer : UINT;
    algoritms_AutoPns_status : UDINT;
    algoritms_AutoTen_status : UDINT;
    algoritms_Remont_status : UDINT;
    algoritms_TestProtection_status : UDINT;
    algoritms_autoNu_NotHasRezervNU : BOOL;
    algoritms_autoNu_status : UDINT;
    algoritms_Pusk_SEC_faza_reactor_Top : UDINT;
    algoritms_Pusk_SEC_faza_reactor_Error : UDINT;
    algoritms_Pusk_SEC_faza_reactor_Start : UDINT;
    algoritms_Pusk_SEC_faza_reactor_status : UDINT;
    algoritms_Pusk_SEC_faza_chastotny_Top : UDINT;
    algoritms_Pusk_SEC_faza_chastotny_Error : UDINT;
    algoritms_Pusk_SEC_faza_chastotny_Start : UDINT;
    algoritms_Pusk_SEC_faza_chastotny_status : UDINT;
    algoritms_Prov_opressovka_ALG_Top : UDINT;
    algoritms_Prov_opressovka_ALG_Error : UDINT;
    algoritms_Prov_opressovka_ALG_Start : UDINT;
    algoritms_Prov_opressovka_ALG_status : UDINT;
    algoritms_Prov_PMS_ALG_Top : UDINT;
    algoritms_Prov_PMS_ALG_Error : UDINT;
    algoritms_Prov_PMS_ALG_Start : UDINT;
    algoritms_Prov_PMS_ALG_status : UDINT;
    algoritms_Pusk_TH_faza_Top : UDINT;
    algoritms_Pusk_TH_faza_Error : UDINT;
    algoritms_Pusk_TH_faza_Start : UDINT;
    algoritms_Pusk_TH_faza_status : UDINT;
    algoritms_Pusk_F_faza2_Top : UDINT;
    algoritms_Pusk_F_faza2_Error : UDINT;
    algoritms_Pusk_F_faza2_Start : UDINT;
    algoritms_Pusk_F_faza2_status : UDINT;
    algoritms_Pusk_F_faza1_Top : UDINT;
    algoritms_Pusk_F_faza1_Error : UDINT;
    algoritms_Pusk_F_faza1_Start : UDINT;
    algoritms_Pusk_F_faza1_status : UDINT;
    algoritms_puskOilSystem_Error : UDINT;
    algoritms_puskOilSystem_Start : UDINT;
    algoritms_puskOilSystem_Top : UDINT;
    algoritms_puskOilSystem_status : UDINT;
    algoritms_testIm_status : UDINT;
    algoritms_vibegPNS_Error : UDINT;
    algoritms_vibegPNS_Start : UDINT;
    algoritms_vibegPNS_Top : UDINT;
    algoritms_vibegPNS_algContinue_status : UDINT;
    algoritms_vibegPNS_status : UDINT;
    algoritms_vibegPNS_waitVibeg_timer : UINT;
    protectManager_protectionInRemont : BOOL;
    algManager : struct_AlgoritmsManager;
    protectManager : struct_ProtectionsManager;
    NotHasRezervNU : BOOL;
    AlgTimers : struct_AlgTimers;
    AlgQuestions : AlgoritmsQuestions;
    algoritms_Apusk_Error : UDINT;
    algoritms_Apusk_Start : UDINT;
    algoritms_Apusk_Top : UDINT;
    algoritms_Apusk_status : UDINT;
    algoritms_RingToLine_Error : UDINT;
    algoritms_RingToLine_Start : UDINT;
    algoritms_RingToLine_Top : UDINT;
    algoritms_RingToLine_status : UDINT;
    algoritms_ao_Error : UDINT;
    algoritms_ao_Start : UDINT;
    algoritms_ao_Top : UDINT;
    algoritms_ao_status : UDINT;
    algoritms_ao_waitKran_timer : UINT;
    algoritms_engineRun_BreakPuskTimer_timer : UINT;
    algoritms_engineRun_Error : UDINT;
    algoritms_engineRun_Start : UDINT;
    algoritms_engineRun_Top : UDINT;
    algoritms_engineRun_status : UDINT;
    algoritms_filling_BreakPuskTimer_timer : UINT;
    algoritms_filling_Error : UDINT;
    algoritms_filling_Start : UDINT;
    algoritms_filling_Top : UDINT;
    algoritms_filling_status : UDINT;
    algoritms_filling_waitAfterKran4_timer : UINT;
    algoritms_filling_waitAfterKran5_timer : UINT;
    algoritms_no_Error : UDINT;
    algoritms_no_Start : UDINT;
    algoritms_no_Top : UDINT;
    algoritms_no_status : UDINT;
    algoritms_no_waitCloseKran_timer : UINT;
    algoritms_ppu_Error : UDINT;
    algoritms_ppu_Start : UDINT;
    algoritms_ppu_Top : UDINT;
    algoritms_ppu_status : UDINT;
    algoritms_puskK_Error : UDINT;
    algoritms_puskK_Start : UDINT;
    algoritms_puskK_Top : UDINT;
    algoritms_puskK_questionFilling_status : UDINT;
    algoritms_puskK_questionUnload_status : UDINT;
    algoritms_puskK_status : UDINT;
    algoritms_autoNu_Start : UDINT;
    algoritms_autoNu_Error : UDINT;
    algoritms_autoNu_Top : UDINT;
    algoritms_AutoAvom_Start : UDINT;
    algoritms_AutoAvom_Error : UDINT;
    algoritms_AutoAvom_Top : UDINT;
    algoritms_puskK_wait720_timer : UINT;
    algoritms_puskOilSystem_BreakPuskTimer_Poil_timer : UINT;
    algoritms_puskOilSystem_BreakPuskTimer_dPmg_timer : UINT;
    algoritms_testPms_BreakTest_timer : UINT;
    algoritms_testPms_Error : UDINT;
    algoritms_testPms_Start : UDINT;
    algoritms_testPms_Top : UDINT;
    algoritms_testPms_algContinue_status : UDINT;
    algoritms_testPms_status : UDINT;
    algoritms_testdPmg_BreakTest_timer : UINT;
    algoritms_testdPmg_Error : UDINT;
    algoritms_testdPmg_Start : UDINT;
    algoritms_testdPmg_Top : UDINT;
    algoritms_testdPmg_algContinue_status : UDINT;
    algoritms_testdPmg_status : UDINT;
  END_VAR

  (* OPC Set - algoritms. Запись текущих состояний тэгов _______________________________________________________*)

  algManager_Mode := algManager.mode;

  protectManager_protectionInRemont:= protectManager.protectionInRemont;

  algoritms_autoNu_NotHasRezervNU:= NotHasRezervNU;

  algoritms_no_Start	:= DWORD_TO_UDINT(algoritms.no.Start);
  algoritms_no_Error	:= DWORD_TO_UDINT(algoritms.no.Error);
  algoritms_no_Top	:= DWORD_TO_UDINT(algoritms.no.Top);
  algoritms_no_status	:= DWORD_TO_UDINT(algoritms.no.status);
  algoritms_no_waitCloseKran_timer	:= AlgTimers.NO_waitCloseKran;

  algoritms_ao_Start	:= DWORD_TO_UDINT(algoritms.ao.Start);
  algoritms_ao_Error	:= DWORD_TO_UDINT(algoritms.ao.Error);
  algoritms_ao_Top	:= DWORD_TO_UDINT(algoritms.ao.Top);
  algoritms_ao_status	:= DWORD_TO_UDINT(algoritms.ao.status);
  algoritms_ao_waitKran_timer	:= AlgTimers.AO_waitKran;

  algoritms_vibegPNS_Start		:= DWORD_TO_UDINT(algoritms.vibegPNS.Start);
  algoritms_vibegPNS_Error		:= DWORD_TO_UDINT(algoritms.vibegPNS.Error);
  algoritms_vibegPNS_Top		:= DWORD_TO_UDINT(algoritms.vibegPNS.Top);
  algoritms_vibegPNS_status		:= DWORD_TO_UDINT(algoritms.vibegPNS.status);
  algoritms_vibegPNS_waitVibeg_timer	:= AlgTimers.vibegPNS_Timer;
  algoritms_vibegPNS_algContinue_status	:= DWORD_TO_UDINT(AlgQuestions.vibegPNS_algContinue.status);

  algoritms_testPms_Start		:= DWORD_TO_UDINT(algoritms.testPms.Start);
  algoritms_testPms_Error		:= DWORD_TO_UDINT(algoritms.testPms.Error);
  algoritms_testPms_Top		:= DWORD_TO_UDINT(algoritms.testPms.Top);
  algoritms_testPms_status		:= DWORD_TO_UDINT(algoritms.testPms.status);
  algoritms_testPms_algContinue_status	:= DWORD_TO_UDINT(AlgQuestions.testPms_algContinue.status);
  algoritms_testPms_BreakTest_timer	:= AlgTimers.testPms_BreakTest;

  algoritms_testdPmg_Start		:= DWORD_TO_UDINT(algoritms.testdPmg.Start);
  algoritms_testdPmg_Error		:= DWORD_TO_UDINT(algoritms.testdPmg.Error);
  algoritms_testdPmg_Top		:= DWORD_TO_UDINT(algoritms.testdPmg.Top);
  algoritms_testdPmg_status		:= DWORD_TO_UDINT(algoritms.testdPmg.status);
  algoritms_testdPmg_algContinue_status	:= DWORD_TO_UDINT(AlgQuestions.testdPmg_algContinue.status);
  algoritms_testdPmg_BreakTest_timer	:= AlgTimers.testdPmg_BreakTest;

  algoritms_testIm_status	:= DWORD_TO_UDINT(algoritms.testIm.status);

  algoritms_ppu_status	:= DWORD_TO_UDINT(algoritms.ppu.status);
  algoritms_ppu_Start	          := DWORD_TO_UDINT(algoritms.ppu.Start);
  algoritms_ppu_Error	          := DWORD_TO_UDINT(algoritms.ppu.Error);
  algoritms_ppu_Top	          := DWORD_TO_UDINT(algoritms.ppu.Top);

  algoritms_puskOilSystem_status			:= DWORD_TO_UDINT(algoritms.puskOilSystem.status);
  algoritms_puskOilSystem_Start				:= DWORD_TO_UDINT(algoritms.puskOilSystem.Start);
  algoritms_puskOilSystem_Error				:= DWORD_TO_UDINT(algoritms.puskOilSystem.Error);
  algoritms_puskOilSystem_Top				:= DWORD_TO_UDINT(algoritms.puskOilSystem.Top);
  algoritms_puskOilSystem_BreakPuskTimer_Poil_timer	          := AlgTimers.puskOilSystem_BreakPuskTimer_Poil;

  algoritms_engineRun_status			:= DWORD_TO_UDINT(algoritms.engineRun.status);
  algoritms_engineRun_Start			:= DWORD_TO_UDINT(algoritms.engineRun.Start);
  algoritms_engineRun_Error			:= DWORD_TO_UDINT(algoritms.engineRun.Error);
  algoritms_engineRun_Top			:= DWORD_TO_UDINT(algoritms.engineRun.Top);
  algoritms_engineRun_BreakPuskTimer_timer	:= AlgTimers.engineRun_BreakPuskTimer;

  algoritms_filling_status		:= DWORD_TO_UDINT(algoritms.filling.status);
  algoritms_filling_Start		:= DWORD_TO_UDINT(algoritms.filling.Start);
  algoritms_filling_Error		:= DWORD_TO_UDINT(algoritms.filling.Error);
  algoritms_filling_Top		:= DWORD_TO_UDINT(algoritms.filling.Top);
  algoritms_filling_BreakPuskTimer_timer	:= AlgTimers.filling_BreakPuskTimer;
  algoritms_filling_waitAfterKran4_timer	:= AlgTimers.filling_waitAfterKran4;
  algoritms_filling_waitAfterKran5_timer	:= AlgTimers.filling_waitAfterKran5;

  algoritms_RingToLine_status	:= DWORD_TO_UDINT(algoritms.RingToLine.status);
  algoritms_RingToLine_Start	:= DWORD_TO_UDINT(algoritms.RingToLine.Start);
  algoritms_RingToLine_Error	:= DWORD_TO_UDINT(algoritms.RingToLine.Error);
  algoritms_RingToLine_Top	:= DWORD_TO_UDINT(algoritms.RingToLine.Top);

  algoritms_AutoPns_status	:= DWORD_TO_UDINT(algoritms.AutoPns.status);
  algoritms_AutoPns_OnTimer	:= AlgTimers.AutoPns_OnTimer;
  algoritms_AutoPns_OffTimer	:= AlgTimers.AutoPns_OffTimer;

  algoritms_autoNu_status	:= DWORD_TO_UDINT(algoritms.autoNu.status);
  algoritms_autoNu_Start	:= DWORD_TO_UDINT(algoritms.autoNu.Start);
  algoritms_autoNu_Error	:= DWORD_TO_UDINT(algoritms.autoNu.Error);
  algoritms_autoNu_Top	:= DWORD_TO_UDINT(algoritms.autoNu.Top);

  algoritms_AutoAvom_status	:= DWORD_TO_UDINT(algoritms.AutoAvom.status);
  algoritms_AutoAvom_Start	:= DWORD_TO_UDINT(algoritms.AutoAvom.Start);
  algoritms_AutoAvom_Error	:= DWORD_TO_UDINT(algoritms.AutoAvom.Error);
  algoritms_AutoAvom_Top	:= DWORD_TO_UDINT(algoritms.AutoAvom.Top);

  algoritms_Pusk_F_faza1_status	:= DWORD_TO_UDINT(algoritms.Pusk_F_faza1.status);
  algoritms_Pusk_F_faza1_Start	:= DWORD_TO_UDINT(algoritms.Pusk_F_faza1.Start);
  algoritms_Pusk_F_faza1_Error	:= DWORD_TO_UDINT(algoritms.Pusk_F_faza1.Error);
  algoritms_Pusk_F_faza1_Top	:= DWORD_TO_UDINT(algoritms.Pusk_F_faza1.Top);

  algoritms_Pusk_F_faza2_status	:= DWORD_TO_UDINT(algoritms.Pusk_F_faza2.status);
  algoritms_Pusk_F_faza2_Start	:= DWORD_TO_UDINT(algoritms.Pusk_F_faza2.Start);
  algoritms_Pusk_F_faza2_Error	:= DWORD_TO_UDINT(algoritms.Pusk_F_faza2.Error);
  algoritms_Pusk_F_faza2_Top	:= DWORD_TO_UDINT(algoritms.Pusk_F_faza2.Top);

  algoritms_Pusk_TH_faza_status	:= DWORD_TO_UDINT(algoritms.Pusk_TH_faza.status);
  algoritms_Pusk_TH_faza_Start	:= DWORD_TO_UDINT(algoritms.Pusk_TH_faza.Start);
  algoritms_Pusk_TH_faza_Error	:= DWORD_TO_UDINT(algoritms.Pusk_TH_faza.Error);
  algoritms_Pusk_TH_faza_Top	:= DWORD_TO_UDINT(algoritms.Pusk_TH_faza.Top);

  algoritms_Prov_PMS_ALG_status	:= DWORD_TO_UDINT(algoritms.Prov_PMS_ALG.status);
  algoritms_Prov_PMS_ALG_Start	:= DWORD_TO_UDINT(algoritms.Prov_PMS_ALG.Start);
  algoritms_Prov_PMS_ALG_Error	:= DWORD_TO_UDINT(algoritms.Prov_PMS_ALG.Error);
  algoritms_Prov_PMS_ALG_Top	:= DWORD_TO_UDINT(algoritms.Prov_PMS_ALG.Top);

  algoritms_Prov_opressovka_ALG_status	:= DWORD_TO_UDINT(algoritms.Prov_opressovka_ALG.status);
  algoritms_Prov_opressovka_ALG_Start	:= DWORD_TO_UDINT(algoritms.Prov_opressovka_ALG.Start);
  algoritms_Prov_opressovka_ALG_Error	:= DWORD_TO_UDINT(algoritms.Prov_opressovka_ALG.Error);
  algoritms_Prov_opressovka_ALG_Top	:= DWORD_TO_UDINT(algoritms.Prov_opressovka_ALG.Top);

  algoritms_Pusk_SEC_faza_chastotny_status	:= DWORD_TO_UDINT(algoritms.Pusk_SEC_faza_chastotny.status);
  algoritms_Pusk_SEC_faza_chastotny_Start	:= DWORD_TO_UDINT(algoritms.Pusk_SEC_faza_chastotny.Start);
  algoritms_Pusk_SEC_faza_chastotny_Error	:= DWORD_TO_UDINT(algoritms.Pusk_SEC_faza_chastotny.Error);
  algoritms_Pusk_SEC_faza_chastotny_Top	:= DWORD_TO_UDINT(algoritms.Pusk_SEC_faza_chastotny.Top);

  algoritms_Pusk_SEC_faza_reactor_status	:= DWORD_TO_UDINT(algoritms.Pusk_SEC_faza_reactor.status);
  algoritms_Pusk_SEC_faza_reactor_Start	:= DWORD_TO_UDINT(algoritms.Pusk_SEC_faza_reactor.Start);
  algoritms_Pusk_SEC_faza_reactor_Error	:= DWORD_TO_UDINT(algoritms.Pusk_SEC_faza_reactor.Error);
  algoritms_Pusk_SEC_faza_reactor_Top	:= DWORD_TO_UDINT(algoritms.Pusk_SEC_faza_reactor.Top);

  algoritms_Remont_status	:= DWORD_TO_UDINT(algoritms.Remont.status);

  algoritms_AutoTen_status	:= DWORD_TO_UDINT(algoritms.AutoTen.status);
END_FUNCTION_BLOCK

FUNCTION_BLOCK fb_OilPump
  VAR_INPUT
    statOn : BOOL;
    statOff : BOOL;
    statOn_reliability : BOOL;
    statOff_reliability : BOOL;
  END_VAR
  VAR_IN_OUT
    StrSw : struct_OilPump;
  END_VAR
  VAR_INPUT
    inNs : TYPE_ReliableBit;
    inAccident : TYPE_ReliableBit;
    inLocal : TYPE_ReliableBit;
    inDistance : TYPE_ReliableBit;
    inBreakCmdOn : TYPE_ReliableBit;
    inBreakCmdOff : TYPE_ReliableBit;
  END_VAR
  VAR
    onInit : BOOL          := FALSE;
    _statOn : BOOL;
    _statOff : BOOL;
    getSdvig : BOOL;
    lastOnStatus : BYTE;
    cmd : BYTE;
    source : BYTE;
    lastCmd : BYTE;
    source_for_Status : BYTE;
    cmd_for_Status : BYTE;
    command_error_for_Status : BYTE;
    _sunpackerCommand : fb_sunpackerCommand;
    _statusDualInput : TYPE_statusDualInput;
    _commandDualInput : TYPE_commandDualInput;
    _commandErrorTimer : BOOL;
    resetErrorTimer : BOOL;
    _changWithoutCommand : BOOL;
    errorCMDTimer : TON;
    sdvigReset : TON;
    _errorReset : TON;
    outputsSets : TOF;
  END_VAR
  VAR_IN_OUT
    cmdOn : BOOL;
    cmdOff : BOOL;
  END_VAR

  IF NOT onInit THEN
  IF StrSw.ISVALIDREF_cmdOn XOR StrSw.ISVALIDREF_cmdOff THEN
  	IF 	StrSw.ISVALIDREF_cmdOn THEN
  		lastCmd:= 2; (*baseCmdOff*)
  	ELSE
  		lastCmd:= 1; (*baseCmdOn*)
  	END_IF;
  END_IF;
  onInit:=TRUE;
  END_IF;

  (* ---- Если управление с ВУ заблокировано, то в ИМ передаем команду из алгоритма ---- *)
  IF StrSw.inOpcCommandsDisabled THEN
  	StrSw.inCommand := StrSw.inCommand_Alg;
  ELSE (* иначе передаем команду с АРМа*)
  	StrSw.inCommand := StrSw.inCommand_ARM;
  END_IF;

  (* ---- Формирование состояния механизма ---- *)

  IF (StrSw.ISVALIDREF_statOn) OR (StrSw.ISVALIDREF_statOff) THEN
  	IF (StrSw.ISVALIDREF_statOn) AND (StrSw.ISVALIDREF_statOff) THEN
  	StrSw.reliability:= statOn_reliability AND statOff_reliability;
  		_statOn  := statOn;
  		_statOff := statOff;
  	ELSIF (StrSw.ISVALIDREF_statOn) THEN
                       StrSw.reliability:= statOn_reliability;
  		_statOn  := statOn;
  		_statOff := NOT statOn;
  	ELSIF (StrSw.ISVALIDREF_statOff) THEN
  		 StrSw.reliability:= statOff_reliability;
  		_statOn  := NOT statOff;
  		_statOff :=statOff;
  	END_IF;

  	IF StrSw.reliability THEN
  		IF _statOn AND NOT _statOff 		THEN 	StrSw.onStatus := _statusDualInput.STATUS_ON;
  		ELSIF _statOff AND NOT _statOn 	THEN 	StrSw.onStatus := _statusDualInput.Status_OFF;
  		ELSIF NOT _statOn AND NOT _statOff 	THEN 	StrSw.onStatus := _statusDualInput.STATUS_TRANSITIONAL;
  		ELSE					StrSw.onStatus := _statusDualInput.STATUS_ERROR;
                      END_IF;

  	ELSE
  		StrSw.onStatus := _statusDualInput.STATUS_NOTDEFINED;

  	END_IF;
  ELSE
  	CASE BYTE_TO_INT(lastCmd) OF
  		(*baseCmdOn*) 1: StrSw.onStatus  := _statusDualInput.STATUS_ON;
  		(*baseCmdOff*) 2: StrSw.onStatus  := _statusDualInput.STATUS_OFF;

  	ELSE
  		 StrSw.onStatus := _statusDualInput.STATUS_NOTDEFINED;

  	END_CASE;
  END_IF;

  StrSw.Accident := inAccident.value AND inAccident.reliability;
  StrSw.Ns := inNs.value AND inNs.reliability;
  StrSw.Local := inLocal.value AND inLocal.reliability;
  StrSw.Distance := inDistance.value AND inDistance.reliability;
  StrSw.OpcCommandsDisabled := StrSw.inOpcCommandsDisabled;

  StrSw.Blocked:=StrSw.Accident OR StrSw.Local OR StrSw.breakCmdOn OR StrSw.breakCmdOff OR StrSw.inBlocked;

  StrSw.Rezervny:=NOT StrSw.Osnovnoy;

  (* ---- Формирование признака сдвига ---- *)

  getSdvig := FALSE;
  IF (StrSw.ISVALIDREF_cmdOn OR StrSw.ISVALIDREF_cmdOff) AND NOT StrSw.Local THEN
  	IF NOT (StrSw.CmdOn OR StrSw.CmdOff) THEN
                       IF (lastOnStatus <> StrSw.onStatus AND
  		(StrSw.onStatus <> _statusDualInput.STATUS_NOTDEFINED AND
                       StrSw.onStatus <> _statusDualInput.STATUS_ERROR)     AND
  		(lastOnStatus <> _statusDualInput.STATUS_NOTDEFINED   AND
                       lastOnStatus <> _statusDualInput.STATUS_ERROR))
                      THEN
  			getSdvig   := TRUE;
  		END_IF;
  	END_IF;
  END_IF;

  IF getSdvig THEN StrSw.sdvig:= TRUE; END_IF;

  sdvigReset(IN:=StrSw.sdvig, PT:=T#15S);

  IF sdvigReset.Q THEN StrSw.sdvig:=FALSE; END_IF;

  lastOnStatus := StrSw.onStatus;

  (* ---- Распаковка команды ---- *)
  _sunpackerCommand(command := StrSw.inCommand);
  	cmd := _sunpackerCommand.cmd;
  	source := _sunpackerCommand.source;

  (* ---- Обработка команды ---- *)
  IF cmd <> 0 AND lastCmd <> cmd and (((NOT StrSw.opcCommandsDisabled) AND source > 0) OR source = 0) then
  	CASE BYTE_TO_INT(cmd) OF
  	(*cmd_on*) 1 :
  			IF  StrSw.ISVALIDREF_cmdOn THEN StrSw.CmdOn := TRUE;
  				IF StrSw.ISVALIDREF_cmdOff THEN StrSw.CmdOff := FALSE; END_IF;
  			ELSIF  StrSw.ISVALIDREF_cmdOff THEN StrSw.CmdOff := FALSE;  END_IF;
  			errorCMDTimer(IN := false);
  			_commandErrorTimer := true;
  			StrSw.lastCmdIsOn := true;
  	(*cmd_off*) 2 :
  			IF StrSw.ISVALIDREF_cmdOff THEN StrSw.CmdOff := TRUE;
  				IF StrSw.ISVALIDREF_cmdOn THEN StrSw.CmdOn := FALSE; END_IF;
  			ELSIF StrSw.ISVALIDREF_cmdOn THEN StrSw.CmdOn := FALSE; END_IF;
  			errorCMDTimer(IN := false);

  			_commandErrorTimer := true;
  			StrSw.lastCmdIsOn := false;
  	(*cmd_reset*) 3 :    IF StrSw.ISVALIDREF_statOn OR StrSw.ISVALIDREF_statOff THEN
  			StrSw.CmdOn := FALSE;
  			StrSw.CmdOff := FALSE;
                                lastCmd := 0;
  			_commandErrorTimer := false;
  			StrSw.lastCmdIsOn := false;
                                 END_IF;
  	END_CASE;
  	source_for_Status := source;
  	cmd_for_Status := cmd;
  	command_error_for_Status := 0;
  END_IF;

  lastCmd := cmd;
  errorCMDTimer(In := _commandErrorTimer, PT :=T#10s);

  (* ---- алгоритм  для команды ВКЛючить ---- *)
  IF (StrSw.onStatus = _statusDualInput.STATUS_ON) and StrSw.lastCmdIsOn then
  	IF StrSw.ISVALIDREF_cmdOn AND StrSw.ISVALIDREF_cmdOff then  StrSw.cmdOn := false; END_IF;

  	 errorCMDTimer(In := false);
  	 _commandErrorTimer := false;
  	 cmd_for_Status := 0;
  	 source_for_Status := 0;
  END_IF;

  (* ---- off ---- *)
  IF (StrSw.onStatus = _statusDualInput.STATUS_OFF) and (NOT StrSw.lastCmdIsOn) then
  	IF StrSw.ISVALIDREF_cmdOn AND StrSw.ISVALIDREF_cmdOff then  StrSw.cmdOff := false; END_IF;

  	 errorCMDTimer(In := false);
  	 _commandErrorTimer := false;
  	 cmd_for_Status := 0;
  	 source_for_Status := 0;
  END_IF;

  (* ---- ошибка исполнения команды ---- *)
  if errorCMDTimer.Q and (cmd_for_Status <> 0) then
  	command_error_for_Status :=  cmd_for_Status;
  	_commandErrorTimer := false;
  	StrSw.CmdOn := false;
  	StrSw.CmdOff := false;
  	lastCmd := 0;
  end_if;

  (* ---- сброс ошибки команды ---- *)
  StrSw.CommandFault := command_error_for_Status <> 0;
  _errorReset(IN := command_error_for_Status <> 0, PT := T#5S);
  IF _errorReset.Q THEN
  	cmd_for_Status := 0;
  	source_for_Status := 0;
  	command_error_for_Status := 0;
  END_IF;

  outputsSets(in := (StrSw.ISVALIDREF_cmdOn and StrSw.cmdOn ) OR (StrSw.ISVALIDREF_cmdOff and StrSw.cmdOff), PT := T#2S);
  	IF NOT outputsSets.Q THEN
  		StrSw.BreakCmdOn := inBreakCmdOn._inversed AND inBreakCmdOn.reliability AND StrSw.ISVALIDREF_inBreakCmdOn;
  		StrSw.BreakCmdOff := inBreakCmdOff._inversed AND inBreakCmdOff.reliability AND StrSw.ISVALIDREF_inBreakCmdOff;
  	END_IF;

  cmdOn := StrSw.cmdOn;
  cmdOff:= StrSw.cmdOff;

  (* ---- формирование зашифрованного статуса для АРМа ---- *)
  StrSw.status := shl(BYTE_TO_DWORD(source_for_Status), 29)
  		OR shl(BYTE_TO_DWORD(cmd_for_Status), 26)
  		OR shl(BYTE_TO_DWORD(command_error_for_Status), 23)
  		OR shl(bool_to_DWORD(StrSw.sdvig), 22)
  		OR shl(bool_to_DWORD(StrSw.OpcCommandsDisabled), 21)
                      OR shl(bool_to_DWORD(StrSw.lastCmdIsOn), 14)
                      OR shl(BOOL_TO_DWORD(StrSw.BreakCmdOff), 13)
  		OR shl(BOOL_TO_DWORD(StrSw.BreakCmdOn), 12)
  		OR shl(BOOL_TO_DWORD(StrSw.Distance), 6)
  		OR shl(BOOL_TO_DWORD(StrSw.Local), 5)
  		OR shl(BOOL_TO_DWORD(StrSw.Ns), 4)
                  	OR shl(BOOL_TO_DWORD(StrSw.Accident ),3)
  		OR BYTE_TO_DWORD(StrSw.onStatus);
END_FUNCTION_BLOCK

FUNCTION_BLOCK Prov_K
  VAR_IN_OUT
    StrAlg : struct_Alg;
  END_VAR
  VAR
    F1_1_start : struct_PhaseAlgoritm;
    F1_2_start : struct_PhaseAlgoritm;
    F3_start : struct_PhaseAlgoritm;
    F4_Start : struct_PhaseAlgoritm;
    Start_Prov_Pusk : struct_Question;
    F4_Start_Q : struct_Question;
    fb_F1_1_start : fb_ph_algoritm;
    fb_F1_2_start : fb_ph_algoritm;
    fb_F3_start : fb_ph_algoritm;
    fb_F4_Start : fb_ph_Kran;
    algoritms : AlgoritmsConfig;
    fb_Start_Prov_Pusk : fb_Question;
    fb_F4_Start_Q : fb_Question;
    fb_kran4Open : fb_ph_Kran;
    fb_kran5Close : fb_ph_Kran;
    fb_kran4Close : fb_ph_Kran;
    fb_timer10 : fb_ph_Timer;
    fb_P_vh_vyh_more_zad : fb_ph_algoritm;
    fb_Zapoln_Norm : fb_ph_algoritm;
    fb_First_Step : fb_ph_algoritm;
    fb_Opressovka_Start : fb_Question;
    fb_PNS_NU_ON_Ask : fb_Question;
    fb_Zapolnit_kontur : fb_Question;
    onInit : BOOL;
  END_VAR
  VAR_EXTERNAL
    Im : ImConfig;
    ai : AiConfig;
  END_VAR
  VAR
    _sunpackerCommand : fb_sunpackerCommand;
    source : BYTE;
    cmd : BYTE;
    _statusDualInput : TYPE_statusDualInput;
    lastCmd : BYTE;
    _Answers : TYPE_Answers;
  END_VAR
  VAR_EXTERNAL
    ModeGpa : TYPE_ModeGpa;
    algManager : struct_AlgoritmsManager;
  END_VAR
  VAR
    cmd_for_Status : BYTE;
    source_for_Status : BYTE;
    command_error_for_Status : BYTE;
    resetCmdTimer : TON;
    waitReset : TON;
    resetCmdTimerPriznak : BOOL;
    _statusAi : TYPE_StatusAi;
    protections : ProtectionsConfig;
  END_VAR

  IF NOT onInit THEN
      fb_F1_1_start(phaseNumber:=1, act:=_run);
      fb_F1_2_start(phaseNumber:=2, act:=_run);
      fb_F3_start(phaseNumber:=3, act:=_run);
      fb_F4_Start(phaseNumber:=4, act:=_on);
      Start_Prov_Pusk.AnswerVariants:=_Answers.ANS_YES + _Answers.ANS_NO;
      F4_Start_Q.AnswerVariants:=_Answers.ANS_YES;
      onInit:=TRUE;
  END_IF;

  fb_F1_1_start(StrPh:=F1_1_start, alg := algoritms.Pusk_F_faza1);
  fb_F1_2_start(StrPh:=F1_2_start, alg := algoritms.Pusk_F_faza2);
  fb_F3_start(StrPh:=F3_start, alg := algoritms.Pusk_TH_faza);
  fb_F4_Start(StrPh:=F4_Start, Im:=Im.Kran6);
  fb_Start_Prov_Pusk(StrQ:=Start_Prov_Pusk);
  fb_F4_Start_Q(StrQ:=F4_Start_Q);

  StrAlg.CanRun := StrAlg.inCanRun;
  StrAlg.OpcCommandsDisabled := StrAlg.inOpcCommandsDisabled;

  IF StrAlg.isRuning THEN
      IF NOT F1_1_start.start THEN
  	askQuestion(Start_Prov_Pusk);
      END_IF;
      IF Start_Prov_Pusk.answer = _Answers.ANS_YES THEN
  	(*algoritms.F1_1.CanRun :=TRUE;*)
  	runPhase(F1_1_start);
  	resetQuestion(Start_Prov_Pusk);
  	(*algManager.setMode(nMode:=ModeGpa.MODE_PUSKK);*)
      ELSIF	Start_Prov_Pusk.answer=_Answers.ANS_NO THEN
  		resetQuestion(Start_Prov_Pusk);
  		(*algoritms.F1_1.CanRun :=FALSE;*)
      END_IF;
      IF F1_1_start.top THEN
  	(*algoritms.F1_2.CanRun :=TRUE;*)
  	runPhase(F1_2_start);
      END_IF;
      IF 	F1_2_start.top (*AND algoritms.ppu.ppuThird*)THEN
  	(*algoritms.F3.CanRun :=TRUE;*)
  	runPhase(F3_start);
      END_IF;
      IF F3_start.top AND (*algoritms.ppu.ppuForth AND*) NOT F4_Start.start  THEN
  	askQuestion(F4_Start_Q);
      ELSE
  	resetQuestion(F4_Start_Q);
      END_IF;
      IF F4_Start_Q.answer = _Answers.ANS_YES THEN
  	resetQuestion(F4_Start_Q);
  	(*algoritms.F4.CanRun :=TRUE;*)
  	runPhase(F4_Start);
      END_IF;
  END_IF;

  _sunpackerCommand(command := StrAlg.inCommand);
  	source := _sunpackerCommand.source;
  	cmd := _sunpackerCommand.cmd;

  IF cmd <> 0 AND lastCmd <> cmd AND (((NOT StrAlg.opcCommandsDisabled) AND source > 0) OR source = 0) then
  	CASE BYTE_TO_INT(cmd) OF
  		(*cm dRun*) 1: 	IF (StrAlg.CanRun) THEN
  					StrAlg.isRuning := TRUE;
  					StrAlg.isEnded := FALSE;
  					StrAlg.hasError := FALSE;
  					(*****************       OnRun       *****************)
                                                    algManager.nMode:=ModeGpa.MODE_PUSK_FIRST_FAZA2;

                                                    (*runPhase(timer120);
                                                    runPhase(timer5);
                                                    runPhase(Shup);
                                                    resetAiProtection(protections.dPmaslo_gaz);
                                                    resetDiProtection(protections.dPmaslo_gaz_less100);*)

  					cmd_for_Status := cmd;
  					source_for_Status := source;
  					command_error_for_Status := 0;
  				ELSE
  					StrAlg.isRuning := FALSE;
  					StrAlg.isEnded := FALSE;
  					StrAlg.hasError := FALSE;

  					cmd_for_Status := 0;
  					source_for_Status := source;
  					command_error_for_Status := cmd;
  				END_IF;
  		(*cmdReset*) 2: 	StrAlg.isRuning := FALSE;
  				StrAlg.isEnded := FALSE;
  				StrAlg.hasError 	:= FALSE;

                                           (*****************       OnReset       *****************)
                                          waitReset(IN:=FALSE);
                                          StrAlg.inCanRun:=FALSE;

                                          (*resetPhase(timer5);
                                          resetPhase(Shup);
                                          resetPhase(timer120);
                                          resetPhase(Net_Chast);
                                          resetPhase(mvOn);
                                          resetPhase(pGNSmore04);
                                          resetPhase(gotov_K_zagruzke);
                                          resetPhase(dPmg_Top);
                                          resetPhase(AutoPNS_Start);*)

                                          StrAlg.inOpcCommandsDisabled:=FALSE;

  				cmd_for_Status := cmd;
  				source_for_Status := source;
  				command_error_for_Status := 0;
  	END_CASE;
  	resetCmdTimer(IN := false);
  	resetCmdTimerPriznak := TRUE;
  END_IF;
  lastCmd := cmd;

  resetCmdTimer(IN := resetCmdTimerPriznak, PT := T#5S);
  IF resetCmdTimer.Q THEN
  	resetCmdTimerPriznak := FALSE;
  	source_for_Status := 0;
  	cmd_for_Status := 0;
  	command_error_for_Status := 0;
  END_IF;

  (*StrAlg.Start:= OPC_Control.startStatus
              OR Pms_more_50.startStatus
              OR Pms_more_300.startStatus
              OR dPmg_more_100.startStatus
              OR P_zad.startStatus
              OR kran5Open.startStatus
              OR kran4Open.startStatus
              OR kran5Close.startStatus
              OR kran4Close.startStatus
              OR timer10.startStatus
              OR P_vh_vyh_more_zad.startStatus
              OR Zapoln_Norm.startStatus
              OR First_Step.startStatus;

  StrAlg.Top :=  OPC_Control.topStatus
              OR Pms_more_50.topStatus
              OR Pms_more_300.topStatus
              OR dPmg_more_100.topStatus
              OR P_zad.topStatus
              OR kran5Open.topStatus
              OR kran4Open.topStatus
              OR kran5Close.topStatus
              OR kran4Close.topStatus
              OR timer10.topStatus
              OR P_vh_vyh_more_zad.topStatus
              OR Zapoln_Norm.topStatus
              OR First_Step.topStatus;

  StrAlg.Error :=  OPC_Control.errorStatus
              OR Pms_more_50.errorStatus
              OR Pms_more_300.errorStatus
              OR dPmg_more_100.errorStatus
              OR P_zad.errorStatus
              OR kran5Open.errorStatus
              OR kran4Open.errorStatus
              OR kran5Close.errorStatus
              OR kran4Close.errorStatus
              OR timer10.errorStatus
              OR P_vh_vyh_more_zad.errorStatus
              OR Zapoln_Norm.errorStatus
              OR First_Step.errorStatus;*)

  (*TODO: TYPE PROGRAM CODE HERE*)
  StrAlg.status :=  SHL(BYTE_TO_DWORD(source_for_Status), 29)
  			OR SHL(BYTE_TO_DWORD(cmd_for_Status), 26)
  			OR SHL(BYTE_TO_DWORD(command_error_for_Status), 23)
  			OR SHL(BOOL_TO_DWORD(StrAlg.OpcCommandsDisabled ), 21)
  			OR SHL(BOOL_TO_DWORD(StrAlg.hasError),4)
  			OR SHL(BOOL_TO_DWORD(StrAlg.CanRun),2)
  			OR SHL(BOOL_TO_DWORD(StrAlg.isEnded),1)
  			OR BOOL_TO_DWORD(StrAlg.isRuning);
END_FUNCTION_BLOCK

FUNCTION_BLOCK Prov_dP_mg
  VAR_IN_OUT
    StrAlg : struct_Alg;
  END_VAR
  VAR
    nu1Off : struct_PhaseAlgoritm;
    nu2Off : struct_PhaseAlgoritm;
    pnsOff : struct_PhaseAlgoritm;
    timer120 : struct_PhaseAlgoritm;
    dPmg_less_100 : struct_PhaseAlgoritm;
    nu1On : struct_PhaseAlgoritm;
    nu2On : struct_PhaseAlgoritm;
    pnsOn : struct_PhaseAlgoritm;
    Error_Alg : struct_PhaseAlgoritm;
    dPmg_more_100 : struct_PhaseAlgoritm;
    fb_nu1Off : fb_ph_OilPump;
    fb_nu2Off : fb_ph_OilPump;
    fb_pnsOff : fb_ph_Switch;
    fb_timer120 : fb_ph_Timer;
    fb_dPmg_less_100 : fb_ph_algoritm;
    fb_nu1On : fb_ph_OilPump;
    fb_nu2On : fb_ph_OilPump;
    fb_pnsOn : fb_ph_Switch;
    fb_Error_Alg : fb_ph_algoritm;
    fb_dPmg_more_100 : fb_ph_algoritm;
    onInit : BOOL;
  END_VAR
  VAR_EXTERNAL
    Im : ImConfig;
    ai : AiConfig;
  END_VAR
  VAR
    _sunpackerCommand : fb_sunpackerCommand;
    source : BYTE;
    cmd : BYTE;
    _statusDualInput : TYPE_statusDualInput;
    lastCmd : BYTE;
    _Answers : TYPE_Answers;
  END_VAR
  VAR_EXTERNAL
    ModeGpa : TYPE_ModeGpa;
    algManager : struct_AlgoritmsManager;
  END_VAR
  VAR
    cmd_for_Status : BYTE;
    source_for_Status : BYTE;
    command_error_for_Status : BYTE;
    resetCmdTimer : TON;
    waitReset : TON;
    resetCmdTimerPriznak : BOOL;
  END_VAR

  IF NOT onInit THEN
      fb_nu1Off(phaseNumber:=1, act:=_off);
      fb_nu2Off(phaseNumber:=2, act:=_off);
      fb_pnsOff(phaseNumber:=3, act:=_off);
      fb_timer120(phaseNumber:=4, delay:=T#120S);
      fb_dPmg_less_100(phaseNumber:=5);
      fb_nu1On(phaseNumber:=6, act:=_on);
      fb_nu2On(phaseNumber:=7, act:=_on);
      fb_pnsOn(phaseNumber:=8, act:=_on);
      fb_Error_Alg(phaseNumber:=9);
      fb_dPmg_more_100(phaseNumber:=10);
      onInit:=TRUE;
  END_IF;

  fb_nu1Off(StrPh:=nu1Off, Im:=Im.nu1);
  fb_nu2Off(StrPh:=nu2Off, Im:=Im.nu2);
  fb_pnsOff(StrPh:=pnsOff, Im:=Im.pns);
  fb_timer120(StrPh:=timer120);
  fb_dPmg_less_100(StrPh:=dPmg_less_100);
  fb_nu1On(StrPh:=nu1On, Im:=Im.nu1);
  fb_nu2On(StrPh:=nu2On, Im:=Im.nu2);
  fb_pnsOn(StrPh:=pnsOn, Im:=Im.pns);
  fb_Error_Alg(StrPh:=Error_Alg);
  fb_dPmg_more_100(StrPh:=dPmg_more_100);

  StrAlg.CanRun := StrAlg.inCanRun;
  StrAlg.OpcCommandsDisabled := StrAlg.inOpcCommandsDisabled;

      IF StrAlg.isRuning THEN
      (* kto takoi ask
          IF	NOT nuOff.start THEN
  	    NU_OFF_Ask.ask ();
      END_IF;*)

      (*
      IF	(nu_OFF_Ask.answer=Answers.ANS_YES) THEN
  	    runPhase(nu1Off);
  	    runPhase(nu2Off);
          runPhase(pnsOff);
  	    NU_OFF_Ask.reset ();
  	    runPhase(timer120);
      END_IF;*)

      (*насосы выключены - запуск проверки *)
      IF	nu1Off.top AND nu2Off.top THEN
  	    runPhase(dPmg_less_100);
      END_IF;

      (*проверка перепада маслогаз по аналогу и дискрету*)
      IF	dPmg_less_100.start AND NOT dPmg_less_100.top THEN
          IF 	Im.SingleSignals.dP_maslo_gaz_Less100.Q AND ai.dPmaslo_gaz.value < 150.0 THEN
  	  	    dPmg_less_100.top:=TRUE;
  		    runPhase(nu1On);
              runPhase(nu2On);
              runPhase(pnsOn);
  	    END_IF;
      END_IF;

      IF	Im.nu1.onStatus = _statusDualInput.STATUS_ON OR Im.nu2.onStatus = _statusDualInput.STATUS_ON  AND nu1On.start  AND nu2On.start AND NOT nu1On.top AND NOT nu2On.top THEN
  	    nu1On.top := TRUE;
          nu2On.top := TRUE;
      END_IF;

      (*ошибка завершения по таймеру*)
      IF	timer120.top THEN
  	    Error_Alg.ERROR := TRUE;
      ELSE
  	    Error_Alg.ERROR := FALSE;
      END_IF;

      (*ыва*)
      IF	nu1On.top AND nu2On.top AND pnsOn.top THEN
  	    runPhase(dPmg_more_100);
      END_IF;

      (**)
      IF	dPmg_more_100.start AND NOT dPmg_more_100.top (*AND NOT algoritms.autoNu_1.flag1 OR algoritms.autoNu_1.flag2*) THEN
  	    IF 	NOT Im.SingleSignals.dP_maslo_gaz_Less100.Q AND Im.SingleSignals.dP_maslo_gaz_Less100.status = 1 AND  ai.dPmaslo_gaz.value > 150.0 THEN
      		dPmg_more_100.top :=TRUE;
  		    resetPhase(timer120);
  	    END_IF;
      END_IF;
  END_IF;

  _sunpackerCommand(command := StrAlg.inCommand);
  	source := _sunpackerCommand.source;
  	cmd := _sunpackerCommand.cmd;

  IF cmd <> 0 AND lastCmd <> cmd AND (((NOT StrAlg.opcCommandsDisabled) AND source > 0) OR source = 0) then
  	CASE BYTE_TO_INT(cmd) OF
  		(*cm dRun*) 1: 	IF (StrAlg.CanRun) THEN
  					StrAlg.isRuning := TRUE;
  					StrAlg.isEnded := FALSE;
  					StrAlg.hasError := FALSE;
  					(*****************       OnRun       *****************)
                                                    algManager.nMode:=ModeGpa.MODE_PUSK_FIRST_FAZA2;

                                                    (*runPhase(timer120);
                                                    runPhase(timer5);
                                                    runPhase(Shup);
                                                    resetAiProtection(protections.dPmaslo_gaz);
                                                    resetDiProtection(protections.dPmaslo_gaz_less100);*)

  					cmd_for_Status := cmd;
  					source_for_Status := source;
  					command_error_for_Status := 0;
  				ELSE
  					StrAlg.isRuning := FALSE;
  					StrAlg.isEnded := FALSE;
  					StrAlg.hasError := FALSE;

  					cmd_for_Status := 0;
  					source_for_Status := source;
  					command_error_for_Status := cmd;
  				END_IF;
  		(*cmdReset*) 2: 	StrAlg.isRuning := FALSE;
  				StrAlg.isEnded := FALSE;
  				StrAlg.hasError 	:= FALSE;

                                           (*****************       OnReset       *****************)
                                          waitReset(IN:=FALSE);
                                          StrAlg.inCanRun:=FALSE;

                                          (*resetPhase(timer5);
                                          resetPhase(Shup);
                                          resetPhase(timer120);
                                          resetPhase(Net_Chast);
                                          resetPhase(mvOn);
                                          resetPhase(pGNSmore04);
                                          resetPhase(gotov_K_zagruzke);
                                          resetPhase(dPmg_Top);
                                          resetPhase(AutoPNS_Start);*)

                                          StrAlg.inOpcCommandsDisabled:=FALSE;

  				cmd_for_Status := cmd;
  				source_for_Status := source;
  				command_error_for_Status := 0;
  	END_CASE;
  	resetCmdTimer(IN := false);
  	resetCmdTimerPriznak := TRUE;
  END_IF;
  lastCmd := cmd;

  resetCmdTimer(IN := resetCmdTimerPriznak, PT := T#5S);
  IF resetCmdTimer.Q THEN
  	resetCmdTimerPriznak := FALSE;
  	source_for_Status := 0;
  	cmd_for_Status := 0;
  	command_error_for_Status := 0;
  END_IF;

  StrAlg.Start:= nu1Off.startStatus
              OR nu2Off.startStatus
              OR pnsOff.startStatus
              OR timer120.startStatus
              OR dPmg_less_100.startStatus
              OR nu1On.startStatus
              OR nu2On.startStatus
              OR pnsOn.startStatus;

  StrAlg.Top := nu1Off.topStatus
              OR nu2Off.topStatus
              OR pnsOff.topStatus
              OR timer120.topStatus
              OR dPmg_less_100.topStatus
              OR nu1On.topStatus
              OR nu2On.topStatus
              OR pnsOn.topStatus;

  StrAlg.Error := nu1Off.errorStatus
              OR nu2Off.errorStatus
              OR pnsOff.errorStatus
              OR timer120.errorStatus
              OR dPmg_less_100.errorStatus
              OR nu1On.errorStatus
              OR nu2On.errorStatus
              OR pnsOn.errorStatus;

  (*TODO: TYPE PROGRAM CODE HERE*)
  StrAlg.status :=  SHL(BYTE_TO_DWORD(source_for_Status), 29)
  			OR SHL(BYTE_TO_DWORD(cmd_for_Status), 26)
  			OR SHL(BYTE_TO_DWORD(command_error_for_Status), 23)
  			OR SHL(BOOL_TO_DWORD(StrAlg.OpcCommandsDisabled ), 21)
  			OR SHL(BOOL_TO_DWORD(StrAlg.hasError),4)
  			OR SHL(BOOL_TO_DWORD(StrAlg.CanRun),2)
  			OR SHL(BOOL_TO_DWORD(StrAlg.isEnded),1)
  			OR BOOL_TO_DWORD(StrAlg.isRuning);
END_FUNCTION_BLOCK

FUNCTION_BLOCK proc_Protections_Init
  VAR_INPUT
    init : BOOL;
  END_VAR
  VAR
    stDIp_Ini : fb_DiProtection_Init;
    stAIp_Ini : fb_AiProtection_Init;
    inits : UINT;
  END_VAR
  VAR_INPUT
    initiales : UINT;
  END_VAR
  VAR_EXTERNAL
    protections : ProtectionsConfig;
  END_VAR
  VAR
    _ProtectionTags : TYPE_ProtectionTags;
    _StatusAi : TYPE_StatusAi;
  END_VAR

  inits := 0; (* Флаг необходимости инициализации структур-дескрипторов *)

  (*************************************************Стартовая инициализация DiProtection ***************************************************)
  (* МВ отключен *)
  stDIp_Ini(data_Ini := true, delay:=T#03S, inTag:=_ProtectionTags.AOS, inRunOnStart:=TRUE, str_DIp := protections.Reg_vozb_off);
  inits := inits + BOOL_TO_UINT(stDIp_Ini.Init);

  (* МВ отключен
  stDIp_Ini(data_Ini := true, delay:=T#1S, inTag:=_ProtectionTags.AOS, inRunOnStart:=FALSE, str_DIp := protections.Fail_chastotnii_pusk);
  inits := inits + BOOL_TO_UINT(stDIp_Ini.Init);*)

  (* МВ отключен *)
  stDIp_Ini(data_Ini := true, delay:=T#1S, inTag:=_ProtectionTags.AOS, inRunOnStart:=TRUE, str_DIp := protections.Off_avar_vikluchatel);
  inits := inits + BOOL_TO_UINT(stDIp_Ini.Init);

  (* МВ отключен *)
  stDIp_Ini(data_Ini := true, delay:=T#1S, inTag:=_ProtectionTags.AOS, inRunOnStart:=TRUE, str_DIp := protections.AOKC_SHKC);
  inits := inits + BOOL_TO_UINT(stDIp_Ini.Init);

  (* МВ отключен *)
  stDIp_Ini(data_Ini := true, delay:=T#0S, inTag:=_ProtectionTags.AOS, inRunOnStart:=TRUE, str_DIp := protections.AO_PRU);
  inits := inits + BOOL_TO_UINT(stDIp_Ini.Init);

  (* МВ отключен *)
  stDIp_Ini(data_Ini := true, delay:=T#0S, inTag:=_ProtectionTags.AOS, inRunOnStart:=FALSE, str_DIp := protections.AO_ot_SHU);
  inits := inits + BOOL_TO_UINT(stDIp_Ini.Init);

  (* МВ отключен *)
  stDIp_Ini(data_Ini := true, delay:=T#1S, inTag:=_ProtectionTags.AOS, inRunOnStart:=FALSE, str_DIp := protections.mvOff);
  inits := inits + BOOL_TO_UINT(stDIp_Ini.Init);

  (* МВ отключен *)
  stDIp_Ini(data_Ini := true, delay:=T#10S, inTag:=_ProtectionTags.AOS, inRunOnStart:=TRUE, str_DIp := protections.Kran1_sdvig);
  inits := inits + BOOL_TO_UINT(stDIp_Ini.Init);

  (* МВ отключен *)
  stDIp_Ini(data_Ini := true, delay:=T#10S, inTag:=_ProtectionTags.AOS, inRunOnStart:=TRUE, str_DIp := protections.Kran2_sdvig);
  inits := inits + BOOL_TO_UINT(stDIp_Ini.Init);

  (* МВ отключен *)
  stDIp_Ini(data_Ini := true, delay:=T#20S, inTag:=_ProtectionTags.AOS, inRunOnStart:=TRUE, str_DIp := protections.dPmaslo_gaz_less100);
  inits := inits + BOOL_TO_UINT(stDIp_Ini.Init);

  (*************************************************Стартовая инициализация AiProtection ***************************************************)
  (* Температура переднего опорного подшипника двигателя, т.1 *)
  stAIp_Ini(data_Ini := true, delay:=T#3S, inTag:=_ProtectionTags.AOS, inRunOnStart:=TRUE,
  controlLimit:=_StatusAi.HA, str_AIp := protections.Topornogo_podshipnika_EDT_1);
  inits := inits + BOOL_TO_UINT(stAIp_Ini.Init);

  (* Температура заднего опорного подшипника двигателя, т.2 *)
  stAIp_Ini(data_Ini := true, delay:=T#3S, inTag:=_ProtectionTags.AOS, inRunOnStart:=TRUE,
  controlLimit:=_StatusAi.HA, str_AIp := protections.Toy_podshipnika_EDT_2);
  inits := inits + BOOL_TO_UINT(stAIp_Ini.Init);

  (* Температура подшипника редуктора, т1 *)
  stAIp_Ini(data_Ini := true, delay:=T#3S, inTag:=_ProtectionTags.AOS, inRunOnStart:=TRUE,
  controlLimit:=_StatusAi.HA, str_AIp := protections.Toy_podshipnika_kol_EDT_3);
  inits := inits + BOOL_TO_UINT(stAIp_Ini.Init);

  (* Температура подшипника редуктора, т2 *)
  stAIp_Ini(data_Ini := true, delay:=T#3S, inTag:=_ProtectionTags.AOS, inRunOnStart:=TRUE,
  controlLimit:=_StatusAi.HA, str_AIp := protections.Toy_podshipnika_kol_EDT_4);
  inits := inits + BOOL_TO_UINT(stAIp_Ini.Init);

  (* Температура подшипника редуктора, т3 *)
  stAIp_Ini(data_Ini := true, delay:=T#3S, inTag:=_ProtectionTags.AOS, inRunOnStart:=TRUE,
  controlLimit:=_StatusAi.HA, str_AIp := protections.To_podshipnika_shest_red_EDT_5);
  inits := inits + BOOL_TO_UINT(stAIp_Ini.Init);

  (* Температура подшипника редуктора, т4 *)
  stAIp_Ini(data_Ini := true, delay:=T#3S, inTag:=_ProtectionTags.AOS, inRunOnStart:=TRUE,
  controlLimit:=_StatusAi.HA, str_AIp := protections.To_podshipnika_shest_red_EDT_6);
  inits := inits + BOOL_TO_UINT(stAIp_Ini.Init);

  (* Температура опорного подшипника нагнетателя, т1 *)
  stAIp_Ini(data_Ini := true, delay:=T#3S, inTag:=_ProtectionTags.AOS, inRunOnStart:=TRUE,
  controlLimit:=_StatusAi.HA, str_AIp := protections.To_podshipnika_N_EDT_7);
  inits := inits + BOOL_TO_UINT(stAIp_Ini.Init);

  (* Температура опорного подшипника нагнетателя, т2 *)
  stAIp_Ini(data_Ini := true, delay:=T#3S, inTag:=_ProtectionTags.AOS, inRunOnStart:=TRUE,
  controlLimit:=_StatusAi.HA, str_AIp := protections.To_podshipnika_svob_konca_EDT_8);
  inits := inits + BOOL_TO_UINT(stAIp_Ini.Init);

  (* Температура опорного подшипника нагнетателя, т3 *)
  stAIp_Ini(data_Ini := true, delay:=T#3S, inTag:=_ProtectionTags.AOS, inRunOnStart:=TRUE,
  controlLimit:=_StatusAi.HA, str_AIp := protections.Ty_podshipnika_rab_kol_EDT_9);
  inits := inits + BOOL_TO_UINT(stAIp_Ini.Init);

  (* Температура упорно опорного подшипника нагнетателя, т4 *)
  stAIp_Ini(data_Ini := true, delay:=T#3S, inTag:=_ProtectionTags.AOS, inRunOnStart:=TRUE,
  controlLimit:=_StatusAi.HA, str_AIp := protections.Typornogo_podshipnika_nerab_kolodok_HT_10);
  inits := inits + BOOL_TO_UINT(stAIp_Ini.Init);

  (* Температура газа на выходе нагнетателя *)
  stAIp_Ini(data_Ini := true, delay:=T#3S, inTag:=_ProtectionTags.AOS, inRunOnStart:=TRUE,
  controlLimit:=_StatusAi.HA, str_AIp := protections.Tgaza_na_vyhode_H);
  inits := inits + BOOL_TO_UINT(stAIp_Ini.Init);

  (* Температура газа на выходе нагнетателя *)
  stAIp_Ini(data_Ini := true, delay:=T#3S, inTag:=_ProtectionTags.AOS, inRunOnStart:=TRUE,
  controlLimit:=_StatusAi.HA, str_AIp := protections.Os_sdvig_nagnetatelja_plus);
  inits := inits + BOOL_TO_UINT(stAIp_Ini.Init);

  (* Температура газа на выходе нагнетателя *)
  stAIp_Ini(data_Ini := true, delay:=T#3S, inTag:=_ProtectionTags.AOS, inRunOnStart:=TRUE,
  controlLimit:=_StatusAi.HA, str_AIp := protections.Os_sdvig_nagnetatelja_minus);
  inits := inits + BOOL_TO_UINT(stAIp_Ini.Init);

  (* Температура газа на выходе нагнетателя *)
  stAIp_Ini(data_Ini := true, delay:=T#3S, inTag:=_ProtectionTags.AOS, inRunOnStart:=TRUE,
  controlLimit:=_StatusAi.HA, str_AIp := protections.Pgaza_na_vyhode_nagnetatelia_GPA_STOP);
  inits := inits + BOOL_TO_UINT(stAIp_Ini.Init);

  (* Температура газа на выходе нагнетателя *)
  stAIp_Ini(data_Ini := true, delay:=T#3S, inTag:=_ProtectionTags.AOS, inRunOnStart:=TRUE,
  controlLimit:=_StatusAi.HA, str_AIp := protections.Pgaza_na_vhode_nagnetatelia_GPA_STOP);
  inits := inits + BOOL_TO_UINT(stAIp_Ini.Init);

  (* Температура газа на выходе нагнетателя *)
  stAIp_Ini(data_Ini := true, delay:=T#3S, inTag:=_ProtectionTags.AOS, inRunOnStart:=TRUE,
  controlLimit:=_StatusAi.HA, str_AIp := protections.Pgaza_na_vyhode_nagnetatelia);
  inits := inits + BOOL_TO_UINT(stAIp_Ini.Init);

  (* Температура газа на выходе нагнетателя *)
  stAIp_Ini(data_Ini := true, delay:=T#20S, inTag:=_ProtectionTags.AOS, inRunOnStart:=TRUE,
  controlLimit:=_StatusAi.HA, str_AIp := protections.dPmaslo_gaz);
  inits := inits + BOOL_TO_UINT(stAIp_Ini.Init);

  (* Температура газа на выходе нагнетателя *)
  stAIp_Ini(data_Ini := true, delay:=T#16S, inTag:=_ProtectionTags.AOS, inRunOnStart:=TRUE,
  controlLimit:=_StatusAi.HA, str_AIp := protections.Pmaslo_sm_nizkoe);
  inits := inits + BOOL_TO_UINT(stAIp_Ini.Init);

  (* Температура газа на выходе нагнетателя *)
  stAIp_Ini(data_Ini := true, delay:=T#16S, inTag:=_ProtectionTags.AOS, inRunOnStart:=TRUE,
  controlLimit:=_StatusAi.HA, str_AIp := protections.Pmaslo_sm_vysokoe);
  inits := inits + BOOL_TO_UINT(stAIp_Ini.Init);

   (* Температура газа на выходе нагнетателя *)
  stAIp_Ini(data_Ini := true, delay:=T#3S, inTag:=_ProtectionTags.AOS, inRunOnStart:=TRUE,
  controlLimit:=_StatusAi.HA, str_AIp := protections.Vibro_skorost_OPED_T1);
  inits := inits + BOOL_TO_UINT(stAIp_Ini.Init);

   (* Температура газа на выходе нагнетателя *)
  stAIp_Ini(data_Ini := true, delay:=T#3S, inTag:=_ProtectionTags.AOS, inRunOnStart:=TRUE,
  controlLimit:=_StatusAi.HA, str_AIp := protections.Vibro_skorost_OPED_T2);
  inits := inits + BOOL_TO_UINT(stAIp_Ini.Init);

   (* Температура газа на выходе нагнетателя *)
  stAIp_Ini(data_Ini := true, delay:=T#3S, inTag:=_ProtectionTags.AOS, inRunOnStart:=TRUE,
  controlLimit:=_StatusAi.HA, str_AIp := protections.Vibro_skorost_OYP_kolesa_ED_T3);
  inits := inits + BOOL_TO_UINT(stAIp_Ini.Init);

   (* Температура газа на выходе нагнетателя *)
  stAIp_Ini(data_Ini := true, delay:=T#3S, inTag:=_ProtectionTags.AOS, inRunOnStart:=TRUE,
  controlLimit:=_StatusAi.HA, str_AIp := protections.Vibro_skorost_OP_kolesa_RH_T4);
  inits := inits + BOOL_TO_UINT(stAIp_Ini.Init);

   (* Температура газа на выходе нагнетателя *)
  stAIp_Ini(data_Ini := true, delay:=T#3S, inTag:=_ProtectionTags.AOS, inRunOnStart:=TRUE,
  controlLimit:=_StatusAi.HA, str_AIp := protections.Vibro_skorost_OP_shesterni_RED_T5);
  inits := inits + BOOL_TO_UINT(stAIp_Ini.Init);

   (* Температура газа на выходе нагнетателя *)
  stAIp_Ini(data_Ini := true, delay:=T#3S, inTag:=_ProtectionTags.AOS, inRunOnStart:=TRUE,
  controlLimit:=_StatusAi.HA, str_AIp := protections.Vibro_skorost_OP_shesterni_RED_T6);
  inits := inits + BOOL_TO_UINT(stAIp_Ini.Init);

   (* Температура газа на выходе нагнетателя *)
  stAIp_Ini(data_Ini := true, delay:=T#3S, inTag:=_ProtectionTags.AOS, inRunOnStart:=TRUE,
  controlLimit:=_StatusAi.HA, str_AIp := protections.Vibro_skorost_OYP_kolesa_ED_T3);
  inits := inits + BOOL_TO_UINT(stAIp_Ini.Init);

   (* Температура газа на выходе нагнетателя *)
  stAIp_Ini(data_Ini := true, delay:=T#3S, inTag:=_ProtectionTags.AOS, inRunOnStart:=TRUE,
  controlLimit:=_StatusAi.HA, str_AIp := protections.Vibro_skorost_OYP_kolesa_ED_T3);
  inits := inits + BOOL_TO_UINT(stAIp_Ini.Init);

   (* Температура газа на выходе нагнетателя *)
  stAIp_Ini(data_Ini := true, delay:=T#3S, inTag:=_ProtectionTags.AOS, inRunOnStart:=TRUE,
  controlLimit:=_StatusAi.HA, str_AIp := protections.Vibro_skorost_OYP_kolesa_ED_T3);
  inits := inits + BOOL_TO_UINT(stAIp_Ini.Init);

  IF init THEN initiales := inits; END_IF;
END_FUNCTION_BLOCK

FUNCTION_BLOCK fb_BaseProtection
  VAR_INPUT
    inSignaling : BOOL;
    inTag : BYTE;
    inRunOnStart : BOOL;
    inCanRun : BOOL;
    inHasError : BOOL;
    inEnded : BOOL;
    inOpcCommandsDisabled : BOOL;
    inCommand : WORD;
  END_VAR
  VAR_OUTPUT
    Tag : BYTE;
    status : DWORD;
    CanRun : BOOL;
    OpcCommandsDisabled : BOOL;
    isRunning : BOOL;
    HasError : BOOL;
    isEnded : BOOL;
    Remont : BOOL;
    Check : BOOL;
    Signaling : BOOL;
    SignalingTP : BOOL;
    RunOnStart : BOOL;
  END_VAR
  VAR
    _sunpackerCommand : fb_sunpackerCommand;
    _ProtectionTags : TYPE_ProtectionTags;
    _signalingTp : TOF;
    source : BYTE;
    cmd : BYTE;
    lastCmd : BYTE;
    source_for_Status : BYTE;
    cmd_for_Status : BYTE;
    command_error_for_Status : BYTE;
    resetCmdTimer : TON;
    resetCmdTimerPriznak : BOOL;
    signalinTimer : TON;
    runOnStart_Trig : R_TRIG;
  END_VAR

  Tag := inTag;
  RunOnStart := inRunOnStart;

  CanRun := inCanRun;
  hasError := inHasError;
  isEnded := inEnded;

  OpcCommandsDisabled := inOpcCommandsDisabled;

  _sunpackerCommand(command := inCommand);
  	source := _sunpackerCommand.source;
  	cmd := _sunpackerCommand.cmd;

  IF cmd <> 0 AND lastCmd <> cmd AND (((NOT opcCommandsDisabled) AND source > 0) OR source = 0) then
  	CASE BYTE_TO_INT(cmd) OF
  		(*cmdRun*) 1: 	IF CanRun AND NOT Remont THEN
  					isEnded := FALSE;
  					hasError 	:= FALSE;
  					isRunning := TRUE;
  					cmd_for_Status := cmd;
  					source_for_Status := source;
  					command_error_for_Status := 0;
  				ELSE
  					isRunning := FALSE;
  					isEnded := FALSE;
  					hasError 	:= FALSE;

  					cmd_for_Status := 0;
  					source_for_Status := source;
  					command_error_for_Status := cmd;
  				END_IF;
  		(*cmdReset*) 2: 	isRunning := FALSE;
  				isEnded := FALSE;
  				hasError 	:= FALSE;
  				inSignaling := FALSE;
  				Check := FALSE;
  				cmd_for_Status := cmd;
  				source_for_Status := source;
  				command_error_for_Status := 0;
  	(*cmd_setRemont*) 4 :	Remont := TRUE;
  				isRunning := FALSE;

  				cmd_for_Status := cmd;
  				source_for_Status := source;
  				command_error_for_Status := 0;
  	(*cmd_resetRemont*) 5 : 	IF inSignaling THEN
  					cmd_for_Status := 0;
  					source_for_Status := 0;
  					command_error_for_Status := cmd;
  				ELSE
  					Remont := FALSE;
  					isRunning := TRUE;

  					cmd_for_Status := cmd;
  					source_for_Status := source;
  					command_error_for_Status := 0;
  				END_IF;
  	(*cmd_setCheck*) 6 : 	Check := TRUE;

  				cmd_for_Status := cmd;
  				source_for_Status := source;
  				command_error_for_Status := 0;
  	END_CASE;
  	resetCmdTimer(IN := false);
  	resetCmdTimerPriznak := TRUE;
  END_IF;
  lastCmd := cmd;

  resetCmdTimer(IN := resetCmdTimerPriznak);
  IF resetCmdTimer.Q THEN
  	resetCmdTimerPriznak := FALSE;
  	source_for_Status := 0;
  	cmd_for_Status := 0;
  	command_error_for_Status := 0;
  END_IF;
